C03662=1154.283,339.501,-77.807,-176.527,8.860,148.763
C03663=1154.278,339.780,-77.845,-176.524,8.864,148.763
C03664=1154.274,340.061,-77.883,-176.521,8.869,148.763
C03665=1154.269,340.309,-77.916,-176.518,8.873,148.764
C03666=1154.266,340.556,-77.950,-176.516,8.876,148.764
C03667=1154.261,340.804,-77.983,-176.513,8.880,148.764
C03668=1154.257,341.051,-78.016,-176.510,8.883,148.764
C03669=1154.254,341.299,-78.051,-176.508,8.887,148.764
C03670=1154.249,341.547,-78.084,-176.505,8.891,148.765
C03671=1154.245,341.795,-78.118,-176.503,8.894,148.765
C03672=1154.241,342.042,-78.151,-176.500,8.898,148.765
C03673=1154.237,342.290,-78.185,-176.498,8.902,148.766
C03674=1154.234,342.537,-78.219,-176.495,8.906,148.766
C03675=1154.229,342.786,-78.253,-176.493,8.909,148.766
C03676=1154.225,343.033,-78.286,-176.491,8.912,148.766
C03677=1154.221,343.280,-78.320,-176.488,8.916,148.767
C03678=1154.217,343.528,-78.353,-176.485,8.920,148.767
C03679=1154.213,343.776,-78.388,-176.483,8.924,148.767
C03680=1154.209,344.024,-78.421,-176.481,8.927,148.767
C03681=1154.205,344.271,-78.455,-176.478,8.931,148.768
C03682=1154.200,344.519,-78.488,-176.475,8.935,148.768
C03683=1154.197,344.767,-78.523,-176.473,8.939,148.768
C03684=1154.193,345.014,-78.557,-176.470,8.942,148.768
C03685=1154.188,345.262,-78.590,-176.468,8.945,148.769
C03686=1154.185,345.510,-78.624,-176.465,8.950,148.769
C03687=1154.181,345.758,-78.658,-176.463,8.953,148.769
C03688=1154.176,346.005,-78.692,-176.460,8.957,148.769
C03689=1154.172,346.252,-78.726,-176.458,8.960,148.770
C03690=1154.169,346.501,-78.760,-176.455,8.965,148.770
C03691=1154.164,346.748,-78.794,-176.453,8.968,148.770
C03692=1154.160,346.996,-78.827,-176.450,8.972,148.771
C03693=1154.157,347.243,-78.861,-176.448,8.975,148.771
C03694=1154.152,347.491,-78.896,-176.445,8.980,148.771
C03695=1154.148,347.738,-78.930,-176.443,8.983,148.771
C03696=1154.144,347.987,-78.964,-176.440,8.987,148.771
C03697=1154.140,348.234,-78.998,-176.438,8.991,148.772
C03698=1154.137,348.481,-79.032,-176.435,8.995,148.772
C03699=1154.133,348.729,-79.066,-176.433,8.998,148.772
C03700=1154.128,348.977,-79.100,-176.430,9.001,148.773
C03701=1154.124,349.224,-79.134,-176.428,9.006,148.773
C03702=1154.121,349.472,-79.168,-176.426,9.009,148.773
C03703=1154.116,349.719,-79.203,-176.423,9.013,148.773
C03704=1154.113,349.967,-79.237,-176.420,9.016,148.774
C03705=1154.108,350.215,-79.271,-176.417,9.020,148.774
C03706=1154.104,350.462,-79.305,-176.416,9.024,148.774
C03707=1154.100,350.711,-79.339,-176.413,9.028,148.775
C03708=1154.096,350.958,-79.373,-176.410,9.031,148.775
C03709=1154.092,351.205,-79.408,-176.407,9.035,148.775
C03710=1154.089,351.453,-79.442,-176.406,9.039,148.775
C03711=1154.084,351.700,-79.476,-176.403,9.043,148.776
C03712=1154.081,351.948,-79.511,-176.400,9.046,148.776
C03713=1154.076,352.196,-79.545,-176.398,9.050,148.776
C03714=1154.073,352.443,-79.579,-176.396,9.054,148.777
C03715=1154.068,352.691,-79.614,-176.393,9.058,148.777
C03716=1154.064,352.939,-79.649,-176.390,9.061,148.777
C03717=1154.061,353.186,-79.683,-176.388,9.066,148.778
C03718=1154.056,353.433,-79.717,-176.386,9.069,148.778
C03719=1154.053,353.681,-79.751,-176.383,9.073,148.778
C03720=1154.048,353.929,-79.786,-176.380,9.077,148.778
C03721=1154.044,354.177,-79.821,-176.378,9.081,148.779
C03722=1154.040,354.424,-79.854,-176.375,9.085,148.779
C03723=1154.036,354.672,-79.889,-176.373,9.088,148.779
C03724=1154.032,354.919,-79.924,-176.370,9.093,148.780
C03725=1154.029,355.167,-79.959,-176.368,9.096,148.780
C03726=1154.024,355.414,-79.993,-176.365,9.100,148.780
C03727=1154.020,355.662,-80.028,-176.363,9.104,148.781
C03728=1154.017,355.909,-80.062,-176.360,9.108,148.781
C03729=1154.013,356.157,-80.097,-176.358,9.111,148.781
C03730=1154.008,356.404,-80.132,-176.355,9.115,148.781
C03731=1154.005,356.652,-80.166,-176.353,9.119,148.782
C03732=1154.001,356.900,-80.201,-176.350,9.123,148.782
C03733=1153.997,357.147,-80.236,-176.348,9.126,148.782
C03734=1153.993,357.395,-80.271,-176.345,9.130,148.783
C03735=1153.989,357.642,-80.305,-176.343,9.135,148.783
C03736=1153.985,357.890,-80.340,-176.341,9.138,148.783
C03737=1153.981,358.137,-80.375,-176.338,9.142,148.784
C03738=1153.977,358.385,-80.410,-176.335,9.146,148.784
C03739=1153.973,358.632,-80.444,-176.333,9.150,148.784
C03740=1153.969,358.880,-80.479,-176.331,9.153,148.784
C03741=1153.965,359.128,-80.514,-176.328,9.157,148.785
C03742=1153.961,359.375,-80.549,-176.325,9.162,148.785
C03743=1153.957,359.623,-80.584,-176.323,9.165,148.785
C03744=1153.954,359.869,-80.619,-176.320,9.169,148.786
C03745=1153.950,360.117,-80.653,-176.318,9.173,148.786
C03746=1153.946,360.366,-80.688,-176.315,9.177,148.786
C03747=1153.941,360.612,-80.723,-176.312,9.181,148.787
C03748=1153.937,360.860,-80.758,-176.311,9.184,148.787
C03749=1153.934,361.108,-80.794,-176.308,9.189,148.787
C03750=1153.929,361.355,-80.828,-176.305,9.193,148.788
C03751=1153.926,361.603,-80.863,-176.303,9.196,148.788
C03752=1153.923,361.850,-80.899,-176.300,9.200,148.788
C03753=1153.918,362.098,-80.933,-176.297,9.205,148.789
C03754=1153.914,362.345,-80.969,-176.295,9.208,148.789
C03755=1153.910,362.593,-81.004,-176.292,9.212,148.789
C03756=1153.906,362.840,-81.039,-176.290,9.217,148.790
C03757=1153.902,363.087,-81.074,-176.287,9.220,148.790
C03758=1153.899,363.336,-81.109,-176.285,9.224,148.790
C03759=1153.894,363.582,-81.144,-176.282,9.228,148.791
C03760=1153.891,363.830,-81.180,-176.280,9.232,148.791
C03761=1153.887,364.078,-81.215,-176.277,9.236,148.791
C03762=1153.882,364.325,-81.250,-176.274,9.240,148.792
C03763=1153.879,364.572,-81.285,-176.273,9.244,148.792
C03764=1153.875,364.820,-81.320,-176.270,9.248,148.792
C03765=1153.870,365.103,-81.360,-176.267,9.252,148.793
C03766=1153.866,365.386,-81.401,-176.264,9.257,148.793
C03767=1153.862,365.669,-81.442,-176.261,9.261,148.794
C03768=1153.857,365.952,-81.481,-176.258,9.266,148.794
C03769=1153.853,366.200,-81.518,-176.256,9.270,148.794
C03770=1153.849,366.447,-81.553,-176.253,9.274,148.795
C03771=1153.845,366.694,-81.588,-176.251,9.278,148.795
C03772=1153.841,366.942,-81.623,-176.249,9.282,148.795
C03773=1153.837,367.190,-81.659,-176.246,9.286,148.796
C03774=1153.834,367.437,-81.694,-176.244,9.290,148.796
C03775=1153.829,367.684,-81.729,-176.241,9.294,148.796
C03776=1153.826,367.931,-81.765,-176.238,9.298,148.797
C03777=1153.822,368.179,-81.801,-176.237,9.302,148.797
C03778=1153.818,368.427,-81.837,-176.234,9.306,148.798
C03779=1153.814,368.674,-81.872,-176.231,9.310,148.798
C03780=1153.810,368.921,-81.907,-176.229,9.314,148.798
C03781=1153.806,369.168,-81.943,-176.227,9.318,148.799
C03782=1153.802,369.416,-81.979,-176.224,9.322,148.799
C03783=1153.799,369.663,-82.014,-176.222,9.326,148.800
C03784=1153.794,369.911,-82.050,-176.220,9.330,148.800
C03785=1153.791,370.159,-82.086,-176.218,9.334,148.801
C03786=1153.786,370.406,-82.121,-176.215,9.338,148.801
C03787=1153.783,370.653,-82.156,-176.213,9.343,148.801
C03788=1153.778,370.901,-82.193,-176.211,9.346,148.802
C03789=1153.775,371.148,-82.228,-176.208,9.350,148.802
C03790=1153.771,371.395,-82.264,-176.206,9.354,148.803
C03791=1153.768,371.643,-82.300,-176.204,9.358,148.803
C03792=1153.763,371.891,-82.336,-176.201,9.363,148.804
C03793=1153.759,372.137,-82.371,-176.200,9.367,148.804
C03794=1153.755,372.385,-82.407,-176.197,9.371,148.805
C03795=1153.752,372.632,-82.442,-176.195,9.375,148.805
C03796=1153.748,372.880,-82.479,-176.193,9.379,148.806
C03797=1153.744,373.127,-82.515,-176.191,9.383,148.806
C03798=1153.740,373.375,-82.550,-176.188,9.387,148.806
C03799=1153.736,373.622,-82.586,-176.187,9.391,148.807
C03800=1153.733,373.869,-82.623,-176.184,9.395,148.808
C03801=1153.729,374.117,-82.658,-176.183,9.399,148.808
C03802=1153.725,374.365,-82.694,-176.180,9.403,148.808
C03803=1153.720,374.611,-82.730,-176.179,9.407,148.809
C03804=1153.717,374.858,-82.766,-176.177,9.411,148.809
C03805=1153.712,375.106,-82.802,-176.175,9.416,148.810
C03806=1153.709,375.354,-82.838,-176.173,9.419,148.811
C03807=1153.705,375.601,-82.874,-176.171,9.423,148.811
C03808=1153.701,375.848,-82.910,-176.169,9.427,148.812
C03809=1153.698,376.095,-82.946,-176.167,9.431,148.812
C03810=1153.693,376.343,-82.982,-176.165,9.435,148.813
C03811=1153.690,376.590,-83.018,-176.163,9.440,148.813
C03812=1153.686,376.838,-83.055,-176.162,9.444,148.814
C03813=1153.682,377.085,-83.090,-176.161,9.447,148.815
C03814=1153.678,377.332,-83.127,-176.159,9.451,148.815
C03815=1153.674,377.580,-83.163,-176.157,9.456,148.816
C03816=1153.670,377.827,-83.200,-176.155,9.460,148.816
C03817=1153.666,378.075,-83.235,-176.154,9.464,148.817
C03818=1153.662,378.322,-83.272,-176.152,9.467,148.818
C03819=1153.659,378.569,-83.308,-176.151,9.471,148.818
C03820=1153.655,378.816,-83.344,-176.149,9.475,148.819
C03821=1153.651,379.064,-83.380,-176.148,9.479,148.819
C03822=1153.647,379.311,-83.417,-176.146,9.483,148.820
C03823=1153.643,379.559,-83.452,-176.145,9.487,148.821
C03824=1153.639,379.806,-83.489,-176.144,9.491,148.821
C03825=1153.635,380.053,-83.525,-176.142,9.495,148.822
C03826=1153.631,380.300,-83.562,-176.141,9.499,148.823
C03827=1153.628,380.547,-83.598,-176.139,9.503,148.823
C03828=1153.623,380.795,-83.634,-176.139,9.506,148.824
C03829=1153.620,381.042,-83.670,-176.137,9.510,148.825
C03830=1153.616,381.290,-83.706,-176.136,9.514,148.826
C03831=1153.612,381.537,-83.743,-176.136,9.517,148.826
C03832=1153.608,381.784,-83.780,-176.134,9.522,148.827
C03833=1153.604,382.032,-83.816,-176.133,9.525,148.828
C03834=1153.601,382.279,-83.852,-176.133,9.529,148.828
C03835=1153.597,382.527,-83.889,-176.132,9.533,148.829
C03836=1153.594,382.773,-83.925,-176.131,9.536,148.830
C03837=1153.589,383.021,-83.962,-176.130,9.540,148.830
C03838=1153.585,383.268,-83.998,-176.129,9.544,148.831
C03839=1153.582,383.515,-84.035,-176.129,9.547,148.832
C03840=1153.577,383.763,-84.071,-176.128,9.551,148.833
C03841=1153.573,384.010,-84.108,-176.127,9.555,148.834
C03842=1153.570,384.257,-84.144,-176.127,9.558,148.834
C03843=1153.566,384.504,-84.181,-176.126,9.561,148.835
C03844=1153.562,384.752,-84.216,-176.126,9.565,148.836
C03845=1153.558,384.999,-84.253,-176.125,9.568,148.837
C03846=1153.554,385.246,-84.290,-176.125,9.572,148.837
C03847=1153.551,385.494,-84.327,-176.124,9.575,148.838
C03848=1153.547,385.741,-84.364,-176.124,9.579,148.839
C03849=1153.543,385.989,-84.400,-176.124,9.582,148.840
C03850=1153.539,386.236,-84.436,-176.123,9.585,148.841
C03851=1153.535,386.483,-84.473,-176.124,9.588,148.842
C03852=1153.531,386.730,-84.510,-176.123,9.592,148.842
C03853=1153.528,386.977,-84.546,-176.123,9.595,148.843
C03854=1153.523,387.225,-84.582,-176.124,9.598,148.844
C03855=1153.519,387.472,-84.619,-176.123,9.601,148.845
C03856=1153.517,387.720,-84.656,-176.124,9.604,148.846
C03857=1153.513,387.967,-84.692,-176.123,9.608,148.846
C03858=1153.508,388.214,-84.729,-176.124,9.610,148.847
C03859=1153.504,388.461,-84.766,-176.124,9.613,148.848
C03860=1153.501,388.708,-84.802,-176.124,9.617,148.849
C03861=1153.497,388.956,-84.839,-176.124,9.620,148.850
C03862=1153.492,389.203,-84.875,-176.124,9.622,148.851
C03863=1153.490,389.451,-84.912,-176.125,9.625,148.851
C03864=1153.486,389.698,-84.949,-176.125,9.628,148.852
C03865=1153.482,389.945,-84.986,-176.126,9.630,148.853
C03866=1153.478,390.192,-85.022,-176.126,9.633,148.854
C03867=1153.474,390.439,-85.059,-176.127,9.636,148.855
C03868=1153.470,390.686,-85.096,-176.127,9.639,148.856
C03869=1153.466,390.973,-85.138,-176.127,9.643,148.857
C03870=1153.461,391.260,-85.181,-176.128,9.646,148.858
C03871=1153.456,391.545,-85.223,-176.128,9.648,148.858
C03872=1153.453,391.832,-85.265,-176.129,9.652,148.860
C03873=1153.449,392.079,-85.302,-176.129,9.654,148.860
C03874=1153.445,392.326,-85.339,-176.130,9.657,148.861
C03875=1153.441,392.573,-85.376,-176.131,9.659,148.862
C03876=1153.437,392.820,-85.412,-176.132,9.662,148.863
C03877=1153.434,393.068,-85.449,-176.132,9.665,148.864
C03878=1153.430,393.315,-85.486,-176.133,9.667,148.864
C03879=1153.426,393.562,-85.523,-176.133,9.670,148.865
C03880=1153.422,393.809,-85.559,-176.134,9.672,148.866
C03881=1153.418,394.056,-85.596,-176.135,9.674,148.867
C03882=1153.414,394.304,-85.633,-176.136,9.676,148.868
C03883=1153.410,394.552,-85.670,-176.136,9.679,148.869
C03884=1153.407,394.799,-85.706,-176.137,9.681,148.869
C03885=1153.403,395.046,-85.742,-176.138,9.684,148.870
C03886=1153.399,395.293,-85.779,-176.139,9.686,148.871
C03887=1153.395,395.541,-85.816,-176.139,9.689,148.872
C03888=1153.391,395.787,-85.852,-176.140,9.691,148.873
C03889=1153.387,396.035,-85.889,-176.141,9.693,148.874
C03890=1153.384,396.283,-85.926,-176.142,9.696,148.875
C03891=1153.379,396.530,-85.963,-176.143,9.698,148.875
C03892=1153.376,396.777,-86.000,-176.144,9.699,148.876
C03893=1153.372,397.024,-86.036,-176.144,9.702,148.877
C03894=1153.368,397.271,-86.073,-176.145,9.704,148.878
C03895=1153.364,397.518,-86.110,-176.146,9.706,148.879
C03896=1153.360,397.766,-86.147,-176.147,9.708,148.879
C03897=1153.357,398.013,-86.184,-176.148,9.711,148.880
C03898=1153.353,398.260,-86.220,-176.149,9.713,148.881
C03899=1153.349,398.507,-86.257,-176.150,9.715,148.882
C03900=1153.345,398.755,-86.294,-176.151,9.717,148.882
C03901=1153.341,399.001,-86.330,-176.152,9.719,148.883
C03902=1153.338,399.249,-86.368,-176.153,9.721,148.884
C03903=1153.334,399.497,-86.405,-176.153,9.723,148.885
C03904=1153.330,399.744,-86.441,-176.154,9.726,148.886
C03905=1153.326,399.991,-86.478,-176.155,9.728,148.887
C03906=1153.322,400.238,-86.515,-176.156,9.730,148.887
C03907=1153.318,400.485,-86.551,-176.157,9.732,148.888
C03908=1153.315,400.733,-86.589,-176.158,9.734,148.889
C03909=1153.311,400.980,-86.625,-176.159,9.735,148.889
C03910=1153.307,401.227,-86.662,-176.160,9.737,148.890
C03911=1153.303,401.475,-86.698,-176.161,9.739,148.891
C03912=1153.299,401.722,-86.735,-176.162,9.741,148.892
C03913=1153.295,401.969,-86.772,-176.163,9.743,148.893
C03914=1153.292,402.217,-86.808,-176.163,9.745,148.893
C03915=1153.288,402.464,-86.845,-176.165,9.747,148.894
C03916=1153.284,402.711,-86.882,-176.166,9.749,148.895
C03917=1153.280,402.958,-86.919,-176.166,9.751,148.896
C03918=1153.275,403.205,-86.956,-176.167,9.753,148.896
C03919=1153.272,403.452,-86.992,-176.168,9.755,148.897
C03920=1153.269,403.700,-87.029,-176.169,9.757,148.898
C03921=1153.265,403.947,-87.066,-176.170,9.759,148.899
C03922=1153.260,404.195,-87.103,-176.171,9.761,148.899
C03923=1153.257,404.441,-87.139,-176.172,9.762,148.900
C03924=1153.253,404.689,-87.176,-176.172,9.764,148.901
C03925=1153.249,404.936,-87.213,-176.174,9.766,148.902
C03926=1153.245,405.184,-87.250,-176.174,9.768,148.902
C03927=1153.241,405.431,-87.287,-176.175,9.770,148.903
C03928=1153.238,405.678,-87.323,-176.176,9.772,148.904
C03929=1153.234,405.925,-87.360,-176.177,9.773,148.904
C03930=1153.230,406.172,-87.397,-176.178,9.776,148.905
C03931=1153.226,406.419,-87.434,-176.179,9.777,148.906
C03932=1153.222,406.667,-87.471,-176.180,9.779,148.907
C03933=1153.219,406.914,-87.507,-176.180,9.781,148.907
C03934=1153.215,407.161,-87.544,-176.181,9.783,148.908
C03935=1153.211,407.409,-87.581,-176.182,9.785,148.909
C03936=1153.207,407.656,-87.618,-176.183,9.787,148.909
C03937=1153.203,407.903,-87.654,-176.183,9.788,148.910
C03938=1153.200,408.151,-87.691,-176.184,9.790,148.911
C03939=1153.196,408.398,-87.728,-176.185,9.792,148.912
C03940=1153.191,408.645,-87.765,-176.186,9.794,148.912
C03941=1153.187,408.892,-87.802,-176.187,9.796,148.913
C03942=1153.184,409.139,-87.838,-176.187,9.797,148.913
C03943=1153.180,409.386,-87.875,-176.188,9.800,148.914
C03944=1153.176,409.634,-87.912,-176.189,9.801,148.915
C03945=1153.172,409.881,-87.949,-176.190,9.803,148.916
C03946=1153.168,410.128,-87.986,-176.190,9.805,148.916
C03947=1153.165,410.375,-88.022,-176.191,9.807,148.917
C03948=1153.161,410.622,-88.059,-176.192,9.808,148.918
C03949=1153.157,410.870,-88.096,-176.193,9.810,148.918
C03950=1153.153,411.118,-88.133,-176.194,9.812,148.919
C03951=1153.149,411.365,-88.170,-176.194,9.814,148.920
C03952=1153.146,411.612,-88.206,-176.195,9.816,148.920
C03953=1153.142,411.859,-88.243,-176.196,9.817,148.921
C03954=1153.138,412.106,-88.280,-176.196,9.819,148.922
C03955=1153.134,412.354,-88.317,-176.196,9.822,148.922
C03956=1153.130,412.601,-88.354,-176.197,9.823,148.923
C03957=1153.127,412.848,-88.390,-176.198,9.825,148.924
C03958=1153.123,413.095,-88.427,-176.199,9.827,148.924
C03959=1153.118,413.342,-88.464,-176.199,9.829,148.925
C03960=1153.114,413.590,-88.501,-176.200,9.830,148.925
C03961=1153.111,413.837,-88.538,-176.201,9.832,148.926
C03962=1153.107,414.084,-88.574,-176.202,9.834,148.927
C03963=1153.103,414.332,-88.611,-176.202,9.836,148.928
C03964=1153.099,414.579,-88.648,-176.203,9.838,148.928
C03965=1153.095,414.826,-88.685,-176.203,9.840,148.929
C03966=1153.093,415.073,-88.722,-176.203,9.842,148.929
C03967=1153.090,415.320,-88.759,-176.204,9.843,148.930
C03968=1153.088,415.568,-88.795,-176.205,9.845,148.931
C03969=1153.087,415.777,-88.826,-176.205,9.847,148.931
C03970=1153.087,415.987,-88.857,-176.206,9.848,148.932
C03971=1153.087,416.196,-88.888,-176.206,9.850,148.932
C03972=1153.087,416.407,-88.919,-176.207,9.852,148.933
C03973=1153.091,416.825,-88.981,-176.207,9.854,148.934
C03974=1153.097,417.243,-89.041,-176.209,9.857,148.935
C03975=1152.676,417.245,-89.089,-176.211,9.868,148.938
C03976=1152.673,417.034,-89.059,-176.210,9.867,148.938
C03977=1152.670,416.824,-89.028,-176.210,9.865,148.937
C03978=1152.669,416.613,-88.997,-176.209,9.864,148.937
C03979=1152.667,416.401,-88.966,-176.209,9.862,148.936
C03980=1152.666,416.190,-88.935,-176.209,9.861,148.936
C03981=1152.666,415.979,-88.904,-176.208,9.859,148.935
C03982=1152.666,415.767,-88.873,-176.208,9.858,148.935
C03983=1152.667,415.556,-88.841,-176.207,9.856,148.934
C03984=1152.669,415.309,-88.805,-176.207,9.854,148.934
C03985=1152.672,415.062,-88.768,-176.206,9.853,148.933
C03986=1152.675,414.815,-88.731,-176.206,9.851,148.932
C03987=1152.679,414.567,-88.695,-176.205,9.849,148.932
C03988=1152.683,414.320,-88.658,-176.204,9.847,148.931
C03989=1152.687,414.073,-88.621,-176.204,9.845,148.930
C03990=1152.690,413.825,-88.584,-176.203,9.843,148.930
C03991=1152.694,413.578,-88.547,-176.203,9.841,148.929
C03992=1152.698,413.331,-88.511,-176.202,9.839,148.928
C03993=1152.702,413.084,-88.474,-176.201,9.838,148.928
C03994=1152.706,412.837,-88.437,-176.200,9.836,148.927
C03995=1152.710,412.589,-88.400,-176.200,9.834,148.926
C03996=1152.713,412.342,-88.363,-176.199,9.832,148.926
C03997=1152.717,412.095,-88.326,-176.198,9.831,148.925
C03998=1152.721,411.847,-88.290,-176.198,9.829,148.924
C03999=1152.725,411.600,-88.253,-176.197,9.827,148.924
C04000=1152.729,411.353,-88.216,-176.197,9.825,148.923
C04001=1152.733,411.105,-88.179,-176.196,9.822,148.922
C04002=1152.736,410.858,-88.142,-176.195,9.821,148.922
C04003=1152.740,410.611,-88.106,-176.195,9.819,148.921
C04004=1152.744,410.364,-88.069,-176.194,9.817,148.920
C04005=1152.748,410.117,-88.032,-176.193,9.815,148.920
C04006=1152.752,409.869,-87.995,-176.192,9.814,148.919
C04007=1152.755,409.622,-87.958,-176.191,9.812,148.918
C04008=1152.759,409.375,-87.922,-176.191,9.810,148.918
C04009=1152.763,409.128,-87.885,-176.190,9.808,148.917
C04010=1152.768,408.880,-87.848,-176.189,9.806,148.916
C04011=1152.772,408.633,-87.811,-176.188,9.804,148.915
C04012=1152.774,408.386,-87.774,-176.188,9.803,148.915
C04013=1152.778,408.138,-87.737,-176.187,9.801,148.914
C04014=1152.783,407.891,-87.701,-176.186,9.799,148.914
C04015=1152.787,407.644,-87.664,-176.185,9.797,148.913
C04016=1152.790,407.397,-87.627,-176.184,9.795,148.912
C04017=1152.794,407.149,-87.590,-176.184,9.794,148.911
C04018=1152.798,406.902,-87.553,-176.183,9.791,148.911
C04019=1152.802,406.655,-87.517,-176.182,9.790,148.910
C04020=1152.806,406.408,-87.480,-176.181,9.788,148.909
C04021=1152.809,406.161,-87.443,-176.180,9.786,148.908
C04022=1152.813,405.914,-87.407,-176.179,9.784,148.908
C04023=1152.817,405.666,-87.369,-176.178,9.782,148.907
C04024=1152.821,405.419,-87.332,-176.177,9.781,148.906
C04025=1152.825,405.171,-87.296,-176.176,9.779,148.906
C04026=1152.828,404.925,-87.259,-176.175,9.777,148.905
C04027=1152.832,404.677,-87.222,-176.175,9.776,148.904
C04028=1152.836,404.430,-87.186,-176.173,9.774,148.903
C04029=1152.840,404.182,-87.148,-176.173,9.772,148.903
C04030=1152.844,403.935,-87.112,-176.172,9.770,148.902
C04031=1152.847,403.688,-87.075,-176.171,9.768,148.901
C04032=1152.852,403.441,-87.038,-176.170,9.766,148.900
C04033=1152.856,403.194,-87.002,-176.169,9.764,148.900
C04034=1152.859,402.946,-86.964,-176.168,9.762,148.899
C04035=1152.862,402.699,-86.928,-176.167,9.760,148.898
C04036=1152.867,402.452,-86.891,-176.166,9.758,148.898
C04037=1152.871,402.205,-86.854,-176.165,9.756,148.897
C04038=1152.875,401.957,-86.817,-176.164,9.754,148.896
C04039=1152.879,401.710,-86.781,-176.163,9.752,148.895
C04040=1152.882,401.463,-86.744,-176.163,9.751,148.895
C04041=1152.886,401.215,-86.707,-176.162,9.749,148.894
C04042=1152.890,400.968,-86.670,-176.160,9.747,148.893
C04043=1152.894,400.721,-86.633,-176.160,9.745,148.892
C04044=1152.898,400.474,-86.597,-176.159,9.742,148.891
C04045=1152.901,400.227,-86.560,-176.158,9.740,148.890
C04046=1152.905,399.979,-86.523,-176.157,9.738,148.890
C04047=1152.909,399.732,-86.486,-176.156,9.736,148.889
C04048=1152.913,399.485,-86.449,-176.155,9.734,148.888
C04049=1152.916,399.238,-86.413,-176.154,9.732,148.888
C04050=1152.920,398.991,-86.376,-176.153,9.730,148.887
C04051=1152.925,398.744,-86.339,-176.152,9.728,148.886
C04052=1152.928,398.496,-86.302,-176.151,9.726,148.885
C04053=1152.932,398.248,-86.265,-176.151,9.724,148.884
C04054=1152.935,398.002,-86.229,-176.150,9.721,148.883
C04055=1152.940,397.754,-86.192,-176.149,9.719,148.883
C04056=1152.944,397.507,-86.155,-176.148,9.717,148.882
C04057=1152.948,397.260,-86.118,-176.147,9.716,148.881
C04058=1152.951,397.012,-86.082,-176.146,9.713,148.880
C04059=1152.955,396.765,-86.045,-176.145,9.711,148.879
C04060=1152.959,396.518,-86.008,-176.144,9.709,148.879
C04061=1152.963,396.271,-85.971,-176.143,9.707,148.878
C04062=1152.967,396.024,-85.934,-176.143,9.704,148.877
C04063=1152.970,395.777,-85.898,-176.142,9.702,148.876
C04064=1152.974,395.529,-85.861,-176.141,9.700,148.875
C04065=1152.978,395.282,-85.824,-176.140,9.697,148.874
C04066=1152.982,395.034,-85.787,-176.139,9.695,148.874
C04067=1152.985,394.788,-85.751,-176.139,9.692,148.873
C04068=1152.989,394.540,-85.714,-176.138,9.690,148.872
C04069=1152.993,394.293,-85.677,-176.137,9.687,148.871
C04070=1152.998,394.046,-85.640,-176.136,9.685,148.870
C04071=1153.000,393.798,-85.604,-176.136,9.682,148.869
C04072=1153.004,393.551,-85.567,-176.135,9.681,148.869
C04073=1153.009,393.303,-85.531,-176.134,9.678,148.868
C04074=1153.013,393.056,-85.494,-176.133,9.676,148.867
C04075=1153.016,392.809,-85.458,-176.133,9.673,148.866
C04076=1153.020,392.562,-85.421,-176.132,9.670,148.865
C04077=1153.024,392.314,-85.384,-176.132,9.668,148.865
C04078=1153.028,392.067,-85.347,-176.131,9.665,148.864
C04079=1153.031,391.820,-85.310,-176.131,9.663,148.863
C04080=1153.035,391.534,-85.267,-176.130,9.660,148.862
C04081=1153.040,391.248,-85.225,-176.129,9.656,148.861
C04082=1153.045,390.961,-85.183,-176.129,9.654,148.860
C04083=1153.049,390.675,-85.140,-176.128,9.651,148.859
C04084=1153.053,390.428,-85.103,-176.127,9.648,148.858
C04085=1153.057,390.181,-85.066,-176.127,9.645,148.857
C04086=1153.060,389.934,-85.030,-176.126,9.642,148.856
C04087=1153.065,389.686,-84.994,-176.127,9.639,148.856
C04088=1153.069,389.439,-84.957,-176.126,9.636,148.855
C04089=1153.072,389.191,-84.920,-176.126,9.633,148.854
C04090=1153.076,388.944,-84.883,-176.126,9.630,148.853
C04091=1153.080,388.697,-84.847,-176.125,9.628,148.852
C04092=1153.084,388.450,-84.810,-176.125,9.625,148.851
C04093=1153.087,388.203,-84.773,-176.125,9.621,148.850
C04094=1153.091,387.956,-84.737,-176.124,9.618,148.850
C04095=1153.096,387.708,-84.700,-176.125,9.615,148.849
C04096=1153.099,387.460,-84.664,-176.124,9.612,148.848
C04097=1153.103,387.213,-84.627,-176.125,9.609,148.847
C04098=1153.107,386.966,-84.590,-176.125,9.606,148.846
C04099=1153.110,386.719,-84.554,-176.125,9.603,148.845
C04100=1153.114,386.472,-84.517,-176.125,9.600,148.845
C04101=1153.118,386.225,-84.480,-176.125,9.596,148.844
C04102=1153.122,385.977,-84.445,-176.125,9.593,148.843
C04103=1153.126,385.730,-84.408,-176.126,9.590,148.842
C04104=1153.130,385.483,-84.371,-176.126,9.587,148.842
C04105=1153.133,385.235,-84.334,-176.126,9.583,148.841
C04106=1153.137,384.988,-84.297,-176.126,9.580,148.840
C04107=1153.141,384.740,-84.261,-176.127,9.576,148.839
C04108=1153.145,384.493,-84.225,-176.127,9.573,148.838
C04109=1153.149,384.246,-84.188,-176.128,9.569,148.838
C04110=1153.153,383.999,-84.151,-176.128,9.566,148.837
C04111=1153.157,383.751,-84.116,-176.129,9.562,148.836
C04112=1153.161,383.504,-84.079,-176.129,9.559,148.835
C04113=1153.165,383.257,-84.042,-176.130,9.555,148.834
C04114=1153.168,383.010,-84.006,-176.131,9.551,148.834
C04115=1153.172,382.762,-83.969,-176.132,9.548,148.833
C04116=1153.175,382.515,-83.933,-176.133,9.544,148.832
C04117=1153.179,382.268,-83.896,-176.133,9.541,148.832
C04118=1153.184,382.020,-83.859,-176.135,9.537,148.831
C04119=1153.187,381.773,-83.824,-176.136,9.532,148.830
C04120=1153.191,381.526,-83.787,-176.137,9.529,148.830
C04121=1153.195,381.279,-83.751,-176.138,9.525,148.829
C04122=1153.199,381.031,-83.714,-176.139,9.521,148.828
C04123=1153.203,380.784,-83.678,-176.140,9.518,148.827
C04124=1153.207,380.536,-83.642,-176.141,9.514,148.827
C04125=1153.211,380.289,-83.605,-176.143,9.510,148.826
C04126=1153.214,380.042,-83.569,-176.144,9.506,148.825
C04127=1153.219,379.794,-83.533,-176.145,9.502,148.825
C04128=1153.222,379.548,-83.497,-176.147,9.498,148.824
C04129=1153.226,379.300,-83.460,-176.148,9.494,148.823
C04130=1153.230,379.053,-83.424,-176.150,9.490,148.823
C04131=1153.234,378.806,-83.387,-176.151,9.486,148.822
C04132=1153.238,378.558,-83.352,-176.152,9.482,148.821
C04133=1153.242,378.311,-83.315,-176.154,9.478,148.821
C04134=1153.245,378.063,-83.279,-176.155,9.474,148.820
C04135=1153.249,377.816,-83.242,-176.157,9.471,148.820
C04136=1153.253,377.569,-83.207,-176.158,9.467,148.819
C04137=1153.257,377.322,-83.170,-176.160,9.462,148.818
C04138=1153.261,377.074,-83.134,-176.162,9.458,148.818
C04139=1153.265,376.827,-83.098,-176.163,9.454,148.817
C04140=1153.269,376.579,-83.062,-176.165,9.451,148.817
C04141=1153.273,376.332,-83.026,-176.167,9.446,148.816
C04142=1153.276,376.085,-82.990,-176.169,9.442,148.815
C04143=1153.280,375.837,-82.954,-176.171,9.439,148.815
C04144=1153.284,375.590,-82.917,-176.173,9.434,148.814
C04145=1153.288,375.342,-82.882,-176.175,9.430,148.814
C04146=1153.292,375.095,-82.846,-176.176,9.427,148.813
C04147=1153.296,374.848,-82.809,-176.179,9.422,148.813
C04148=1153.299,374.600,-82.774,-176.180,9.419,148.812
C04149=1153.304,374.352,-82.738,-176.182,9.414,148.812
C04150=1153.307,374.106,-82.701,-176.184,9.410,148.811
C04151=1153.311,373.858,-82.665,-176.187,9.406,148.811
C04152=1153.315,373.610,-82.630,-176.188,9.402,148.810
C04153=1153.319,373.364,-82.594,-176.191,9.398,148.810
C04154=1153.323,373.116,-82.558,-176.193,9.394,148.809
C04155=1153.327,372.869,-82.522,-176.195,9.390,148.809
C04156=1153.331,372.621,-82.487,-176.197,9.386,148.808
C04157=1153.334,372.374,-82.451,-176.199,9.381,148.808
C04158=1153.338,372.127,-82.414,-176.201,9.378,148.807
C04159=1153.342,371.879,-82.379,-176.203,9.373,148.807
C04160=1153.346,371.632,-82.343,-176.205,9.370,148.806
C04161=1153.350,371.384,-82.307,-176.208,9.365,148.806
C04162=1153.354,371.137,-82.272,-176.210,9.361,148.806
C04163=1153.358,370.889,-82.236,-176.213,9.358,148.805
C04164=1153.361,370.643,-82.200,-176.215,9.353,148.805
C04165=1153.366,370.395,-82.164,-176.217,9.350,148.804
C04166=1153.370,370.147,-82.128,-176.219,9.345,148.804
C04167=1153.373,369.900,-82.093,-176.222,9.341,148.803
C04168=1153.377,369.652,-82.057,-176.224,9.337,148.803
C04169=1153.381,369.406,-82.022,-176.226,9.333,148.803
C04170=1153.385,369.158,-81.986,-176.229,9.329,148.802
C04171=1153.389,368.910,-81.950,-176.231,9.325,148.802
C04172=1153.393,368.663,-81.915,-176.234,9.321,148.801
C04173=1153.396,368.415,-81.879,-176.236,9.317,148.801
C04174=1153.401,368.168,-81.844,-176.238,9.313,148.801
C04175=1153.404,367.921,-81.808,-176.241,9.309,148.800
C04176=1153.409,367.673,-81.772,-176.244,9.305,148.800
C04177=1153.412,367.426,-81.737,-176.246,9.301,148.800
C04178=1153.416,367.178,-81.701,-176.248,9.297,148.799
C04179=1153.421,366.931,-81.667,-176.251,9.292,148.799
C04180=1153.424,366.683,-81.631,-176.253,9.289,148.798
C04181=1153.428,366.436,-81.596,-176.256,9.285,148.798
C04182=1153.432,366.188,-81.560,-176.258,9.280,148.798
C04183=1153.436,365.941,-81.525,-176.261,9.277,148.797
C04184=1153.440,365.658,-81.484,-176.264,9.272,148.797
C04185=1153.445,365.375,-81.443,-176.266,9.267,148.796
C04186=1153.449,365.092,-81.403,-176.269,9.263,148.796
C04187=1153.453,364.809,-81.363,-176.272,9.258,148.796
C04188=1153.458,364.561,-81.328,-176.275,9.254,148.795
C04189=1153.462,364.314,-81.293,-176.277,9.250,148.795
C04190=1153.465,364.066,-81.257,-176.280,9.246,148.795
C04191=1153.469,363.818,-81.222,-176.283,9.242,148.794
C04192=1153.474,363.572,-81.187,-176.285,9.239,148.794
C04193=1153.477,363.324,-81.152,-176.287,9.235,148.794
C04194=1153.481,363.076,-81.117,-176.290,9.230,148.793
C04195=1153.486,362.829,-81.082,-176.292,9.227,148.793
C04196=1153.489,362.582,-81.046,-176.295,9.223,148.793
C04197=1153.493,362.333,-81.011,-176.298,9.218,148.792
C04198=1153.497,362.087,-80.976,-176.300,9.215,148.792
C04199=1153.501,361.839,-80.940,-176.302,9.211,148.792
C04200=1153.505,361.591,-80.906,-176.305,9.207,148.791
C04201=1153.509,361.345,-80.871,-176.308,9.203,148.791
C04202=1153.513,361.096,-80.836,-176.310,9.199,148.791
C04203=1153.516,360.849,-80.801,-176.312,9.196,148.790
C04204=1153.521,360.602,-80.766,-176.315,9.192,148.790
C04205=1153.524,360.354,-80.731,-176.318,9.187,148.790
C04206=1153.528,360.106,-80.696,-176.320,9.184,148.790
C04207=1153.533,359.859,-80.661,-176.323,9.180,148.789
C04208=1153.536,359.611,-80.626,-176.325,9.175,148.789
C04209=1153.540,359.365,-80.591,-176.328,9.172,148.789
C04210=1153.544,359.116,-80.556,-176.330,9.168,148.788
C04211=1153.548,358.868,-80.522,-176.333,9.164,148.788
C04212=1153.552,358.621,-80.486,-176.335,9.160,148.788
C04213=1153.556,358.374,-80.452,-176.338,9.156,148.787
C04214=1153.560,358.126,-80.418,-176.340,9.153,148.787
C04215=1153.564,357.879,-80.382,-176.343,9.149,148.787
C04216=1153.568,357.631,-80.347,-176.345,9.145,148.786
C04217=1153.572,357.383,-80.313,-176.348,9.141,148.786
C04218=1153.575,357.136,-80.278,-176.350,9.138,148.786
C04219=1153.580,356.889,-80.243,-176.353,9.133,148.785
C04220=1153.584,356.640,-80.209,-176.356,9.129,148.785
C04221=1153.587,356.394,-80.174,-176.358,9.126,148.785
C04222=1153.591,356.146,-80.139,-176.360,9.121,148.784
C04223=1153.596,355.898,-80.105,-176.363,9.118,148.784
C04224=1153.600,355.650,-80.070,-176.366,9.114,148.784
C04225=1153.604,355.403,-80.036,-176.368,9.110,148.784
C04226=1153.607,355.156,-80.000,-176.370,9.106,148.783
C04227=1153.612,354.908,-79.966,-176.373,9.103,148.783
C04228=1153.615,354.660,-79.932,-176.375,9.099,148.783
C04229=1153.620,354.413,-79.897,-176.378,9.095,148.782
C04230=1153.624,354.165,-79.862,-176.380,9.091,148.782
C04231=1153.628,353.918,-79.829,-176.383,9.088,148.782
C04232=1153.631,353.670,-79.794,-176.385,9.084,148.781
C04233=1153.635,353.423,-79.760,-176.388,9.080,148.781
C04234=1153.639,353.175,-79.724,-176.390,9.076,148.781
C04235=1153.644,352.928,-79.690,-176.393,9.072,148.780
C04236=1153.647,352.680,-79.656,-176.395,9.069,148.780
C04237=1153.651,352.432,-79.621,-176.398,9.065,148.780
C04238=1153.655,352.185,-79.587,-176.400,9.061,148.780
C04239=1153.659,351.937,-79.552,-176.403,9.057,148.779
C04240=1153.662,351.689,-79.518,-176.405,9.054,148.779
C04241=1153.667,351.442,-79.484,-176.408,9.049,148.779
C04242=1153.672,351.194,-79.450,-176.410,9.046,148.778
C04243=1153.675,350.946,-79.416,-176.413,9.042,148.778
C04244=1153.680,350.699,-79.381,-176.415,9.038,148.778
C04245=1153.683,350.451,-79.347,-176.418,9.034,148.778
C04246=1153.687,350.204,-79.313,-176.420,9.031,148.777
C04247=1153.691,349.956,-79.279,-176.423,9.027,148.777
C04248=1153.695,349.708,-79.244,-176.425,9.023,148.777
C04249=1153.699,349.461,-79.210,-176.428,9.019,148.777
C04250=1153.703,349.213,-79.175,-176.430,9.016,148.776
C04251=1153.707,348.965,-79.142,-176.433,9.012,148.776
C04252=1153.711,348.718,-79.108,-176.435,9.008,148.776
C04253=1153.715,348.470,-79.073,-176.438,9.004,148.775
C04254=1153.719,348.223,-79.039,-176.440,9.001,148.775
C04255=1153.724,347.975,-79.006,-176.443,8.997,148.775
C04256=1153.727,347.727,-78.971,-176.445,8.993,148.775
C04257=1153.731,347.480,-78.937,-176.448,8.989,148.774
C04258=1153.735,347.233,-78.903,-176.450,8.986,148.774
C04259=1153.739,346.984,-78.870,-176.453,8.983,148.774
C04260=1153.743,346.737,-78.835,-176.455,8.978,148.773
C04261=1153.747,346.490,-78.801,-176.458,8.975,148.773
C04262=1153.752,346.241,-78.767,-176.460,8.971,148.773
C04263=1153.755,345.994,-78.733,-176.463,8.968,148.773
C04264=1153.759,345.747,-78.699,-176.466,8.964,148.773
C04265=1153.764,345.499,-78.666,-176.468,8.960,148.772
C04266=1153.767,345.251,-78.631,-176.470,8.956,148.772
C04267=1153.771,345.003,-78.598,-176.473,8.953,148.772
C04268=1153.776,344.756,-78.564,-176.476,8.948,148.771
C04269=1153.780,344.507,-78.530,-176.478,8.945,148.771
C04270=1153.783,344.260,-78.496,-176.481,8.941,148.771
C04271=1153.787,344.013,-78.463,-176.483,8.938,148.771
C04272=1153.792,343.765,-78.429,-176.485,8.934,148.770
C04273=1153.795,343.517,-78.395,-176.488,8.930,148.770
C04274=1153.799,343.269,-78.361,-176.490,8.927,148.770
C04275=1153.804,343.021,-78.328,-176.493,8.923,148.770
C04276=1153.808,342.774,-78.294,-176.495,8.919,148.769
C04277=1153.812,342.527,-78.261,-176.498,8.915,148.769
C04278=1153.816,342.279,-78.226,-176.501,8.912,148.769
C04279=1153.820,342.031,-78.193,-176.503,8.908,148.769
C04280=1153.824,341.784,-78.159,-176.505,8.904,148.768
C04281=1153.828,341.536,-78.126,-176.508,8.901,148.768
C04282=1153.832,341.287,-78.092,-176.511,8.897,148.768
C04283=1153.836,341.040,-78.058,-176.513,8.894,148.768
C04284=1153.840,340.793,-78.025,-176.516,8.890,148.767
C04285=1153.845,340.545,-77.991,-176.518,8.886,148.767
C04286=1153.849,340.297,-77.957,-176.521,8.882,148.767
C04287=1153.853,340.050,-77.924,-176.523,8.879,148.767
C04288=1153.857,339.769,-77.886,-176.526,8.875,148.766
C04289=1153.862,339.490,-77.848,-176.529,8.871,148.766
C04290=1153.866,339.209,-77.810,-176.532,8.866,148.766
C04291=1153.871,338.930,-77.773,-176.535,8.862,148.766
C04292=1153.875,338.682,-77.740,-176.537,8.859,148.765
C04293=1153.879,338.434,-77.706,-176.540,8.855,148.765
C04294=1153.882,338.186,-77.673,-176.542,8.852,148.765
C04295=1153.887,337.938,-77.640,-176.545,8.848,148.765
C04296=1153.890,337.691,-77.606,-176.547,8.844,148.764
C04297=1153.895,337.443,-77.572,-176.550,8.841,148.764
C04298=1153.899,337.195,-77.539,-176.552,8.837,148.764
C04299=1153.904,336.947,-77.506,-176.555,8.834,148.764
C04300=1153.908,336.700,-77.473,-176.558,8.830,148.764
C04301=1153.912,336.452,-77.440,-176.560,8.826,148.763
C04302=1153.916,336.204,-77.406,-176.562,8.823,148.763
C04303=1153.920,335.956,-77.373,-176.565,8.819,148.763
C04304=1153.924,335.708,-77.340,-176.567,8.815,148.763
C04305=1153.927,335.461,-77.307,-176.570,8.811,148.762
C04306=1153.931,335.213,-77.274,-176.572,8.808,148.762
C04307=1153.935,334.965,-77.241,-176.575,8.805,148.762
C04308=1153.940,334.717,-77.208,-176.578,8.801,148.762
C04309=1153.944,334.470,-77.175,-176.580,8.797,148.761
C04310=1153.948,334.222,-77.141,-176.583,8.793,148.761
C04311=1153.952,333.974,-77.108,-176.585,8.790,148.761
C04312=1153.956,333.727,-77.075,-176.587,8.787,148.761
C04313=1153.960,333.479,-77.042,-176.590,8.783,148.761
C04314=1153.964,333.231,-77.009,-176.593,8.779,148.760
C04315=1153.968,332.983,-76.976,-176.595,8.776,148.760
C04316=1153.973,332.736,-76.942,-176.598,8.772,148.760
C04317=1153.976,332.488,-76.910,-176.600,8.769,148.760
C04318=1153.980,332.240,-76.877,-176.603,8.765,148.759
C04319=1153.985,331.992,-76.844,-176.605,8.761,148.759
C04320=1153.989,331.744,-76.811,-176.608,8.758,148.759
C04321=1153.993,331.497,-76.778,-176.611,8.754,148.759
C04322=1153.997,331.249,-76.745,-176.613,8.751,148.759
C04323=1154.001,331.001,-76.713,-176.616,8.748,148.759
C04324=1154.005,330.753,-76.680,-176.619,8.744,148.758
C04325=1154.009,330.505,-76.647,-176.621,8.740,148.758
C04326=1154.013,330.258,-76.614,-176.624,8.736,148.758
C04327=1154.018,330.009,-76.581,-176.626,8.733,148.758
C04328=1154.021,329.762,-76.549,-176.628,8.730,148.758
C04329=1154.025,329.514,-76.515,-176.631,8.726,148.757
C04330=1154.030,329.266,-76.483,-176.634,8.722,148.757
C04331=1154.034,329.018,-76.450,-176.636,8.719,148.757
C04332=1154.037,328.771,-76.417,-176.639,8.715,148.757
C04333=1154.042,328.522,-76.385,-176.641,8.712,148.756
C04334=1154.046,328.275,-76.352,-176.643,8.708,148.756
C04335=1154.049,328.027,-76.320,-176.646,8.704,148.756
C04336=1154.054,327.780,-76.287,-176.649,8.701,148.756
C04337=1154.058,327.532,-76.254,-176.651,8.698,148.756
C04338=1154.062,327.284,-76.222,-176.654,8.694,148.755
C04339=1154.066,327.036,-76.189,-176.657,8.691,148.755
C04340=1154.071,326.788,-76.156,-176.659,8.687,148.755
C04341=1154.074,326.540,-76.124,-176.662,8.683,148.755
C04342=1154.078,326.292,-76.091,-176.664,8.680,148.755
C04343=1154.083,326.044,-76.058,-176.666,8.677,148.755
C04344=1154.086,325.796,-76.026,-176.669,8.673,148.754
C04345=1154.091,325.549,-75.994,-176.672,8.669,148.754
C04346=1154.095,325.301,-75.961,-176.674,8.666,148.754
C04347=1154.099,325.053,-75.929,-176.677,8.662,148.754
C04348=1154.103,324.805,-75.896,-176.680,8.659,148.754
C04349=1154.107,324.557,-75.864,-176.682,8.656,148.754
C04350=1154.111,324.309,-75.831,-176.685,8.652,148.753
C04351=1154.115,324.062,-75.800,-176.687,8.648,148.753
C04352=1154.120,323.814,-75.767,-176.689,8.645,148.753
C04353=1154.123,323.566,-75.735,-176.692,8.641,148.753
C04354=1154.128,323.318,-75.702,-176.695,8.638,148.752
C04355=1154.131,323.070,-75.670,-176.697,8.634,148.752
C04356=1154.136,322.822,-75.637,-176.700,8.631,148.752
C04357=1154.140,322.575,-75.606,-176.703,8.627,148.752
C04358=1154.144,322.326,-75.573,-176.705,8.624,148.752
C04359=1154.148,322.079,-75.541,-176.707,8.621,148.752
C04360=1154.152,321.831,-75.508,-176.710,8.617,148.751
C04361=1154.156,321.583,-75.476,-176.712,8.613,148.751
C04362=1154.161,321.335,-75.444,-176.715,8.610,148.751
C04363=1154.164,321.088,-75.412,-176.718,8.606,148.751
C04364=1154.169,320.839,-75.379,-176.720,8.603,148.751
C04365=1154.172,320.591,-75.348,-176.723,8.600,148.751
C04366=1154.177,320.343,-75.315,-176.725,8.597,148.750
C04367=1154.181,320.095,-75.284,-176.728,8.593,148.750
C04368=1154.185,319.847,-75.252,-176.731,8.589,148.750
C04369=1154.189,319.599,-75.219,-176.733,8.586,148.750
C04370=1154.193,319.352,-75.187,-176.736,8.582,148.750
C04371=1154.197,319.104,-75.155,-176.738,8.579,148.750
C04372=1154.201,318.856,-75.123,-176.741,8.576,148.750
C04373=1154.205,318.608,-75.091,-176.743,8.573,148.749
C04374=1154.210,318.360,-75.059,-176.746,8.569,148.749
C04375=1154.214,318.112,-75.027,-176.748,8.565,148.749
C04376=1154.218,317.864,-74.995,-176.751,8.562,148.749
C04377=1154.223,317.617,-74.963,-176.754,8.558,148.749
C04378=1154.226,317.368,-74.931,-176.756,8.555,148.749
C04379=1154.230,317.120,-74.899,-176.759,8.552,148.748
C04380=1154.234,316.873,-74.868,-176.761,8.548,148.748
C04381=1154.239,316.625,-74.836,-176.764,8.545,148.748
C04382=1154.243,316.377,-74.804,-176.767,8.541,148.748
C04383=1154.247,316.129,-74.772,-176.769,8.538,148.748
C04384=1154.251,315.881,-74.740,-176.771,8.535,148.748
C04385=1154.255,315.632,-74.709,-176.775,8.531,148.748
C04386=1154.260,315.385,-74.677,-176.777,8.528,148.747
C04387=1154.263,315.137,-74.645,-176.779,8.524,148.747
C04388=1154.268,314.889,-74.613,-176.782,8.521,148.747
C04389=1154.272,314.641,-74.581,-176.785,8.517,148.747
C04390=1154.276,314.393,-74.550,-176.787,8.514,148.747
C04391=1154.280,314.146,-74.518,-176.790,8.511,148.747
C04392=1154.285,313.868,-74.483,-176.792,8.507,148.746
C04393=1154.289,313.590,-74.448,-176.796,8.503,148.746
C04394=1154.294,313.313,-74.412,-176.799,8.499,148.746
C04395=1154.299,313.036,-74.376,-176.801,8.496,148.746
C04396=1154.303,312.788,-74.344,-176.804,8.493,148.746
C04397=1154.307,312.540,-74.314,-176.807,8.489,148.746
C04398=1154.311,312.292,-74.282,-176.809,8.485,148.746
C04399=1154.315,312.044,-74.250,-176.812,8.482,148.746
C04400=1154.319,311.796,-74.219,-176.814,8.479,148.745
C04401=1154.323,311.548,-74.187,-176.817,8.475,148.745
C04402=1154.327,311.300,-74.156,-176.819,8.472,148.745
C04403=1154.332,311.051,-74.124,-176.822,8.469,148.745
C04404=1154.336,310.804,-74.093,-176.824,8.465,148.745
C04405=1154.340,310.555,-74.061,-176.827,8.461,148.745
C04406=1154.345,310.308,-74.030,-176.830,8.458,148.745
C04407=1154.348,310.060,-73.998,-176.832,8.455,148.744
C04408=1154.353,309.812,-73.967,-176.835,8.452,148.744
C04409=1154.357,309.564,-73.935,-176.838,8.448,148.744
C04410=1154.361,309.316,-73.905,-176.840,8.445,148.744
C04411=1154.365,309.068,-73.873,-176.843,8.441,148.744
C04412=1154.370,308.820,-73.842,-176.845,8.439,148.744
C04413=1154.373,308.572,-73.810,-176.848,8.435,148.744
C04414=1154.378,308.324,-73.780,-176.851,8.431,148.744
C04415=1154.382,308.076,-73.748,-176.853,8.428,148.744
C04416=1154.386,307.828,-73.717,-176.856,8.425,148.743
C04417=1154.390,307.580,-73.685,-176.858,8.422,148.743
C04418=1154.395,307.332,-73.654,-176.861,8.418,148.743
C04419=1154.399,307.083,-73.623,-176.864,8.415,148.743
C04420=1154.403,306.836,-73.592,-176.866,8.412,148.743
C04421=1154.408,306.588,-73.561,-176.869,8.408,148.743
C04422=1154.411,306.340,-73.529,-176.871,8.405,148.743
C04423=1154.416,306.092,-73.498,-176.874,8.401,148.743
C04424=1154.420,305.843,-73.467,-176.877,8.398,148.742
C04425=1154.424,305.596,-73.436,-176.879,8.395,148.742
C04426=1154.428,305.348,-73.405,-176.882,8.392,148.742
C04427=1154.432,305.100,-73.374,-176.884,8.389,148.742
C04428=1154.436,304.852,-73.343,-176.887,8.385,148.742
C04429=1154.440,304.604,-73.312,-176.890,8.381,148.742
C04430=1154.445,304.356,-73.281,-176.892,8.378,148.742
C04431=1154.449,304.107,-73.250,-176.895,8.375,148.742
C04432=1154.454,303.859,-73.219,-176.897,8.372,148.742
C04433=1154.458,303.612,-73.188,-176.900,8.368,148.742
C04434=1154.461,303.363,-73.157,-176.903,8.365,148.741
C04435=1154.466,303.115,-73.126,-176.905,8.362,148.741
C04436=1154.471,302.867,-73.096,-176.908,8.359,148.741
C04437=1154.475,302.619,-73.064,-176.910,8.355,148.741
C04438=1154.479,302.371,-73.033,-176.913,8.352,148.741
C04439=1154.483,302.124,-73.003,-176.916,8.348,148.741
C04440=1154.487,301.875,-72.972,-176.919,8.345,148.741
C04441=1154.491,301.627,-72.941,-176.921,8.342,148.741
C04442=1154.496,301.379,-72.910,-176.924,8.339,148.741
C04443=1154.499,301.131,-72.880,-176.926,8.336,148.741
C04444=1154.504,300.883,-72.849,-176.929,8.333,148.741
C04445=1154.508,300.635,-72.818,-176.932,8.329,148.740
C04446=1154.512,300.386,-72.787,-176.934,8.326,148.740
C04447=1154.516,300.139,-72.757,-176.937,8.323,148.740
C04448=1154.521,299.891,-72.726,-176.939,8.319,148.740
C04449=1154.525,299.642,-72.695,-176.942,8.316,148.740
C04450=1154.529,299.394,-72.665,-176.944,8.313,148.740
C04451=1154.533,299.146,-72.634,-176.947,8.309,148.740
C04452=1154.537,298.898,-72.603,-176.950,8.306,148.740
C04453=1154.541,298.650,-72.573,-176.952,8.303,148.740
C04454=1154.546,298.402,-72.542,-176.955,8.300,148.740
C04455=1154.551,298.154,-72.511,-176.958,8.297,148.740
C04456=1154.554,297.906,-72.481,-176.960,8.294,148.739
C04457=1154.558,297.658,-72.450,-176.963,8.290,148.739
C04458=1154.563,297.410,-72.419,-176.965,8.287,148.739
C04459=1154.567,297.162,-72.390,-176.968,8.284,148.739
C04460=1154.571,296.913,-72.358,-176.971,8.280,148.739
C04461=1154.575,296.665,-72.328,-176.973,8.277,148.739
C04462=1154.580,296.417,-72.298,-176.976,8.274,148.739
C04463=1154.584,296.170,-72.267,-176.978,8.271,148.739
C04464=1154.588,295.921,-72.237,-176.981,8.267,148.739
C04465=1154.593,295.673,-72.206,-176.984,8.264,148.739
C04466=1154.596,295.425,-72.176,-176.986,8.261,148.739
C04467=1154.601,295.177,-72.145,-176.989,8.258,148.739
C04468=1154.605,294.929,-72.116,-176.991,8.255,148.738
C04469=1154.609,294.680,-72.085,-176.994,8.252,148.739
C04470=1154.613,294.432,-72.055,-176.997,8.248,148.738
C04471=1154.618,294.184,-72.024,-177.000,8.245,148.738
C04472=1154.622,293.936,-71.994,-177.002,8.241,148.738
C04473=1154.627,293.688,-71.964,-177.005,8.238,148.738
C04474=1154.630,293.441,-71.933,-177.008,8.235,148.738
C04475=1154.634,293.192,-71.904,-177.010,8.232,148.738
C04476=1154.639,292.944,-71.873,-177.013,8.229,148.738
C04477=1154.643,292.695,-71.843,-177.015,8.226,148.738
C04478=1154.647,292.447,-71.813,-177.018,8.223,148.738
C04479=1154.651,292.200,-71.782,-177.021,8.219,148.738
C04480=1154.656,291.951,-71.752,-177.024,8.216,148.738
C04481=1154.659,291.703,-71.722,-177.026,8.213,148.738
C04482=1154.664,291.455,-71.692,-177.029,8.210,148.738
C04483=1154.668,291.207,-71.662,-177.031,8.207,148.738
C04484=1154.672,290.958,-71.632,-177.034,8.203,148.738
C04485=1154.677,290.710,-71.601,-177.036,8.200,148.738
C04486=1154.681,290.462,-71.572,-177.039,8.197,148.737
C04487=1154.685,290.214,-71.542,-177.042,8.193,148.737
C04488=1154.690,289.966,-71.512,-177.045,8.190,148.737
C04489=1154.694,289.718,-71.482,-177.047,8.187,148.737
C04490=1154.698,289.470,-71.452,-177.050,8.184,148.737
C04491=1154.702,289.221,-71.422,-177.052,8.181,148.737
C04492=1154.706,288.973,-71.392,-177.055,8.178,148.737
C04493=1154.710,288.725,-71.362,-177.058,8.175,148.737
C04494=1154.714,288.477,-71.332,-177.060,8.172,148.737
C04495=1154.719,288.229,-71.302,-177.063,8.169,148.737
C04496=1154.724,287.954,-71.269,-177.066,8.165,148.737
C04497=1154.729,287.678,-71.236,-177.069,8.162,148.737
C04498=1154.733,287.404,-71.203,-177.072,8.158,148.737
C04499=1154.738,287.128,-71.170,-177.075,8.154,148.737
C04500=1154.742,286.879,-71.140,-177.078,8.151,148.737
C04501=1154.746,286.632,-71.110,-177.080,8.148,148.737
C04502=1154.751,286.383,-71.080,-177.083,8.145,148.737
C04503=1154.755,286.135,-71.051,-177.085,8.142,148.737
C04504=1154.759,285.887,-71.021,-177.088,8.139,148.737
C04505=1154.763,285.639,-70.991,-177.090,8.136,148.736
C04506=1154.767,285.391,-70.961,-177.093,8.133,148.737
C04507=1154.772,285.142,-70.931,-177.096,8.130,148.737
C04508=1154.776,284.894,-70.902,-177.098,8.126,148.736
C04509=1154.781,284.646,-70.873,-177.101,8.123,148.736
C04510=1154.785,284.399,-70.843,-177.104,8.121,148.736
C04511=1154.789,284.150,-70.813,-177.106,8.117,148.736
C04512=1154.793,283.902,-70.784,-177.109,8.113,148.736
C04513=1154.798,283.653,-70.754,-177.112,8.111,148.736
C04514=1154.802,283.405,-70.724,-177.115,8.107,148.736
C04515=1154.807,283.157,-70.695,-177.117,8.104,148.736
C04516=1154.811,282.909,-70.665,-177.120,8.101,148.736
C04517=1154.815,282.660,-70.636,-177.122,8.098,148.736
C04518=1154.819,282.412,-70.606,-177.125,8.095,148.736
C04519=1154.823,282.164,-70.577,-177.128,8.092,148.736
C04520=1154.828,281.916,-70.548,-177.131,8.089,148.736
C04521=1154.832,281.667,-70.518,-177.133,8.086,148.736
C04522=1154.836,281.419,-70.489,-177.136,8.083,148.736
C04523=1154.840,281.171,-70.459,-177.139,8.080,148.736
C04524=1154.845,280.923,-70.430,-177.141,8.077,148.736
C04525=1154.849,280.675,-70.401,-177.144,8.074,148.736
C04526=1154.853,280.427,-70.371,-177.146,8.071,148.736
C04527=1154.857,280.178,-70.342,-177.149,8.068,148.736
C04528=1154.862,279.930,-70.312,-177.152,8.064,148.736
C04529=1154.866,279.682,-70.283,-177.155,8.061,148.736
C04530=1154.870,279.434,-70.253,-177.158,8.058,148.736
C04531=1154.874,279.185,-70.225,-177.160,8.055,148.736
C04532=1154.879,278.937,-70.196,-177.163,8.052,148.736
C04533=1154.883,278.689,-70.166,-177.165,8.049,148.736
C04534=1154.888,278.441,-70.137,-177.168,8.046,148.736
C04535=1154.892,278.192,-70.107,-177.170,8.043,148.736
C04536=1154.896,277.944,-70.078,-177.173,8.040,148.736
C04537=1154.900,277.695,-70.049,-177.176,8.037,148.736
C04538=1154.905,277.448,-70.020,-177.179,8.034,148.736
C04539=1154.909,277.199,-69.990,-177.181,8.030,148.736
C04540=1154.914,276.951,-69.961,-177.184,8.027,148.736
C04541=1154.917,276.703,-69.933,-177.187,8.025,148.736
C04542=1154.921,276.454,-69.903,-177.189,8.022,148.736
C04543=1154.926,276.207,-69.874,-177.192,8.018,148.736
C04544=1154.931,275.958,-69.846,-177.194,8.015,148.736
C04545=1154.935,275.710,-69.816,-177.197,8.012,148.736
C04546=1154.939,275.461,-69.787,-177.200,8.009,148.736
C04547=1154.943,275.213,-69.759,-177.202,8.006,148.736
C04548=1154.948,274.965,-69.729,-177.205,8.003,148.736
C04549=1154.952,274.717,-69.700,-177.208,8.000,148.736
C04550=1154.956,274.468,-69.671,-177.211,7.997,148.736
C04551=1154.961,274.220,-69.642,-177.213,7.994,148.736
C04552=1154.965,273.972,-69.614,-177.216,7.991,148.736
C04553=1154.969,273.724,-69.585,-177.218,7.988,148.736
C04554=1154.974,273.475,-69.556,-177.221,7.985,148.736
C04555=1154.978,273.226,-69.526,-177.224,7.982,148.736
C04556=1154.982,272.979,-69.498,-177.227,7.979,148.736
C04557=1154.986,272.730,-69.469,-177.229,7.976,148.736
C04558=1154.990,272.482,-69.440,-177.232,7.973,148.736
C04559=1154.995,272.233,-69.411,-177.235,7.970,148.736
C04560=1154.999,271.985,-69.383,-177.237,7.967,148.736
C04561=1155.003,271.737,-69.354,-177.240,7.964,148.736
C04562=1155.008,271.488,-69.325,-177.242,7.961,148.736
C04563=1155.012,271.241,-69.297,-177.245,7.958,148.736
C04564=1155.016,270.992,-69.268,-177.248,7.955,148.736
C04565=1155.021,270.744,-69.238,-177.251,7.952,148.736
C04566=1155.025,270.496,-69.211,-177.254,7.949,148.736
C04567=1155.029,270.247,-69.182,-177.256,7.946,148.736
C04568=1155.034,269.999,-69.152,-177.259,7.943,148.736
C04569=1155.038,269.751,-69.125,-177.261,7.940,148.736
C04570=1155.043,269.502,-69.096,-177.264,7.937,148.736
C04571=1155.047,269.254,-69.066,-177.267,7.934,148.736
C04572=1155.051,269.006,-69.039,-177.270,7.931,148.736
C04573=1155.056,268.757,-69.010,-177.272,7.928,148.736
C04574=1155.060,268.510,-68.981,-177.275,7.925,148.736
C04575=1155.064,268.261,-68.953,-177.278,7.922,148.736
C04576=1155.069,268.012,-68.924,-177.280,7.919,148.736
C04577=1155.073,267.764,-68.896,-177.283,7.916,148.736
C04578=1155.077,267.516,-68.867,-177.286,7.913,148.736
C04579=1155.081,267.267,-68.839,-177.289,7.910,148.736
C04580=1155.086,267.019,-68.810,-177.291,7.907,148.736
C04581=1155.090,266.770,-68.782,-177.294,7.904,148.737
C04582=1155.095,266.522,-68.754,-177.297,7.901,148.736
C04583=1155.099,266.274,-68.725,-177.299,7.898,148.736
C04584=1155.103,266.026,-68.696,-177.302,7.895,148.736
C04585=1155.107,265.777,-68.668,-177.305,7.892,148.737
C04586=1155.112,265.529,-68.640,-177.308,7.889,148.737
C04587=1155.116,265.281,-68.612,-177.310,7.886,148.737
C04588=1155.120,265.032,-68.583,-177.313,7.883,148.737
C04589=1155.125,264.784,-68.555,-177.316,7.881,148.737
C04590=1155.129,264.535,-68.526,-177.319,7.878,148.737
C04591=1155.134,264.287,-68.499,-177.321,7.874,148.737
C04592=1155.138,264.038,-68.470,-177.324,7.871,148.737
C04593=1155.142,263.790,-68.442,-177.326,7.869,148.737
C04594=1155.147,263.541,-68.413,-177.329,7.866,148.737
C04595=1155.151,263.294,-68.386,-177.331,7.863,148.737
C04596=1155.155,263.045,-68.358,-177.334,7.860,148.737
C04597=1155.160,262.797,-68.329,-177.337,7.857,148.737
C04598=1155.164,262.548,-68.301,-177.340,7.855,148.737
C04599=1155.169,262.300,-68.273,-177.343,7.852,148.737
C04600=1155.174,262.027,-68.242,-177.346,7.848,148.737
C04601=1155.178,261.753,-68.211,-177.349,7.845,148.737
C04602=1155.183,261.481,-68.180,-177.351,7.842,148.737
C04603=1155.187,261.207,-68.149,-177.354,7.839,148.737
C04604=1155.192,260.958,-68.120,-177.357,7.836,148.737
C04605=1155.196,260.710,-68.093,-177.360,7.833,148.737
C04606=1155.200,260.461,-68.065,-177.363,7.830,148.738
C04607=1155.205,260.213,-68.037,-177.365,7.827,148.738
C04608=1155.209,259.965,-68.009,-177.368,7.824,148.738
C04609=1155.213,259.717,-67.981,-177.371,7.821,148.738
C04610=1155.217,259.468,-67.954,-177.374,7.818,148.738
C04611=1155.222,259.219,-67.925,-177.376,7.815,148.738
C04612=1155.227,258.972,-67.897,-177.379,7.812,148.738
C04613=1155.231,258.723,-67.869,-177.381,7.809,148.738
C04614=1155.235,258.475,-67.842,-177.384,7.806,148.738
C04615=1155.240,258.226,-67.813,-177.387,7.803,148.738
C04616=1155.244,257.978,-67.786,-177.390,7.800,148.738
C04617=1155.248,257.730,-67.758,-177.392,7.798,148.738
C04618=1155.252,257.481,-67.730,-177.395,7.795,148.738
C04619=1155.258,257.232,-67.702,-177.398,7.792,148.738
C04620=1155.261,256.984,-67.674,-177.400,7.789,148.738
C04621=1155.266,256.735,-67.647,-177.403,7.787,148.738
C04622=1155.270,256.487,-67.619,-177.406,7.784,148.738
C04623=1155.274,256.239,-67.591,-177.409,7.781,148.738
C04624=1155.279,255.990,-67.564,-177.411,7.778,148.738
C04625=1155.284,255.742,-67.536,-177.414,7.775,148.739
C04626=1155.288,255.493,-67.508,-177.417,7.772,148.739
C04627=1155.292,255.245,-67.480,-177.419,7.770,148.739
C04628=1155.297,254.997,-67.453,-177.422,7.767,148.739
C04629=1155.301,254.748,-67.425,-177.425,7.764,148.739
C04630=1155.305,254.500,-67.398,-177.427,7.761,148.739
C04631=1155.310,254.252,-67.370,-177.430,7.758,148.739
C04632=1155.314,254.002,-67.343,-177.433,7.755,148.739
C04633=1155.318,253.755,-67.315,-177.436,7.752,148.739
C04634=1155.323,253.506,-67.288,-177.439,7.749,148.739
C04635=1155.326,253.258,-67.260,-177.441,7.746,148.739
C04636=1155.332,253.009,-67.232,-177.444,7.744,148.739
C04637=1155.336,252.761,-67.204,-177.446,7.741,148.739
C04638=1155.341,252.512,-67.177,-177.449,7.738,148.739
C04639=1155.345,252.264,-67.149,-177.452,7.735,148.739
C04640=1155.349,252.015,-67.122,-177.455,7.733,148.740
C04641=1155.354,251.767,-67.095,-177.458,7.730,148.740
C04642=1155.358,251.518,-67.067,-177.461,7.727,148.740
C04643=1155.362,251.270,-67.040,-177.463,7.724,148.740
C04644=1155.367,251.021,-67.013,-177.466,7.722,148.740
C04645=1155.371,250.773,-66.985,-177.468,7.719,148.740
C04646=1155.375,250.524,-66.958,-177.471,7.716,148.740
C04647=1155.379,250.276,-66.931,-177.474,7.713,148.740
C04648=1155.384,250.028,-66.903,-177.477,7.710,148.740
C04649=1155.388,249.780,-66.876,-177.479,7.707,148.740
C04650=1155.392,249.530,-66.849,-177.482,7.704,148.740
C04651=1155.397,249.282,-66.822,-177.485,7.701,148.741
C04652=1155.401,249.034,-66.794,-177.487,7.699,148.741
C04653=1155.406,248.786,-66.767,-177.490,7.696,148.741
C04654=1155.411,248.537,-66.740,-177.493,7.693,148.741
C04655=1155.415,248.288,-66.713,-177.496,7.690,148.741
C04656=1155.419,248.039,-66.686,-177.499,7.688,148.741
C04657=1155.424,247.791,-66.658,-177.502,7.685,148.741
C04658=1155.428,247.543,-66.631,-177.504,7.682,148.741
C04659=1155.432,247.295,-66.604,-177.507,7.680,148.741
C04660=1155.437,247.046,-66.577,-177.509,7.677,148.741
C04661=1155.441,246.797,-66.550,-177.512,7.674,148.742
C04662=1155.446,246.549,-66.523,-177.515,7.671,148.742
C04663=1155.450,246.300,-66.496,-177.518,7.668,148.742
C04664=1155.454,246.052,-66.469,-177.520,7.665,148.742
C04665=1155.459,245.803,-66.442,-177.523,7.663,148.742
C04666=1155.464,245.555,-66.415,-177.525,7.660,148.742
C04667=1155.468,245.306,-66.388,-177.529,7.657,148.742
C04668=1155.472,245.057,-66.361,-177.531,7.654,148.742
C04669=1155.476,244.809,-66.334,-177.534,7.651,148.742
C04670=1155.481,244.561,-66.307,-177.537,7.648,148.742
C04671=1155.486,244.312,-66.280,-177.539,7.646,148.743
C04672=1155.490,244.064,-66.253,-177.542,7.643,148.743
C04673=1155.494,243.815,-66.226,-177.545,7.640,148.743
C04674=1155.499,243.567,-66.199,-177.547,7.637,148.743
C04675=1155.503,243.318,-66.172,-177.551,7.635,148.743
C04676=1155.507,243.070,-66.146,-177.553,7.633,148.743
C04677=1155.512,242.822,-66.119,-177.556,7.630,148.743
C04678=1155.516,242.573,-66.091,-177.558,7.627,148.743
C04679=1155.520,242.324,-66.065,-177.561,7.624,148.743
C04680=1155.525,242.076,-66.038,-177.564,7.621,148.743
C04681=1155.529,241.827,-66.011,-177.566,7.619,148.744
C04682=1155.534,241.579,-65.985,-177.569,7.616,148.744
C04683=1155.538,241.330,-65.958,-177.572,7.613,148.744
C04684=1155.543,241.082,-65.931,-177.575,7.610,148.744
C04685=1155.547,240.833,-65.904,-177.578,7.607,148.744
C04686=1155.551,240.585,-65.877,-177.581,7.605,148.744
C04687=1155.556,240.336,-65.851,-177.583,7.602,148.744
C04688=1155.560,240.088,-65.825,-177.586,7.600,148.745
C04689=1155.565,239.839,-65.797,-177.589,7.597,148.745
C04690=1155.569,239.591,-65.771,-177.592,7.594,148.745
C04691=1155.574,239.342,-65.745,-177.594,7.592,148.745
C04692=1155.578,239.094,-65.718,-177.597,7.589,148.745
C04693=1155.582,238.845,-65.691,-177.599,7.586,148.745
C04694=1155.587,238.596,-65.665,-177.603,7.583,148.745
C04695=1155.591,238.348,-65.638,-177.605,7.580,148.745
C04696=1155.596,238.099,-65.611,-177.608,7.578,148.745
C04697=1155.600,237.850,-65.585,-177.610,7.575,148.745
C04698=1155.605,237.602,-65.558,-177.613,7.572,148.746
C04699=1155.609,237.354,-65.532,-177.616,7.570,148.746
C04700=1155.614,237.105,-65.506,-177.619,7.567,148.746
C04701=1155.618,236.857,-65.479,-177.621,7.565,148.746
C04702=1155.623,236.607,-65.453,-177.624,7.562,148.746
C04703=1155.627,236.359,-65.426,-177.627,7.559,148.746
C04704=1155.632,236.087,-65.398,-177.630,7.556,148.746
C04705=1155.636,235.816,-65.369,-177.633,7.553,148.747
C04706=1155.641,235.544,-65.340,-177.636,7.550,148.747
C04707=1155.646,235.272,-65.312,-177.639,7.548,148.747
C04708=1155.651,235.024,-65.284,-177.642,7.545,148.747
C04709=1155.655,234.775,-65.259,-177.644,7.542,148.747
C04710=1155.660,234.526,-65.232,-177.647,7.539,148.747
C04711=1155.664,234.278,-65.206,-177.649,7.537,148.747
C04712=1155.668,234.029,-65.179,-177.653,7.534,148.748
C04713=1155.673,233.781,-65.153,-177.655,7.531,148.748
C04714=1155.678,233.532,-65.128,-177.658,7.528,148.748
C04715=1155.682,233.284,-65.101,-177.660,7.526,148.748
C04716=1155.686,233.035,-65.075,-177.664,7.524,148.748
C04717=1155.690,232.787,-65.048,-177.666,7.521,148.748
C04718=1155.695,232.538,-65.022,-177.669,7.518,148.748
C04719=1155.700,232.289,-64.996,-177.671,7.516,148.748
C04720=1155.704,232.041,-64.970,-177.675,7.513,148.749
C04721=1155.709,231.792,-64.944,-177.677,7.510,148.749
C04722=1155.713,231.543,-64.918,-177.680,7.508,148.749
C04723=1155.717,231.295,-64.892,-177.682,7.505,148.749
C04724=1155.721,231.046,-64.866,-177.686,7.503,148.749
C04725=1155.726,230.797,-64.840,-177.688,7.500,148.749
C04726=1155.731,230.549,-64.814,-177.691,7.498,148.749
C04727=1155.735,230.301,-64.788,-177.693,7.495,148.750
C04728=1155.740,230.052,-64.761,-177.697,7.492,148.750
C04729=1155.744,229.803,-64.736,-177.699,7.489,148.750
C04730=1155.749,229.554,-64.710,-177.702,7.487,148.750
C04731=1155.753,229.307,-64.684,-177.704,7.484,148.750
C04732=1155.757,229.058,-64.658,-177.708,7.481,148.750
C04733=1155.762,228.809,-64.632,-177.710,7.479,148.751
C04734=1155.766,228.560,-64.606,-177.713,7.476,148.751
C04735=1155.771,228.311,-64.580,-177.716,7.474,148.751
C04736=1155.776,228.063,-64.555,-177.719,7.471,148.751
C04737=1155.780,227.814,-64.529,-177.721,7.469,148.751
C04738=1155.784,227.566,-64.502,-177.724,7.466,148.751
C04739=1155.789,227.317,-64.476,-177.727,7.463,148.752
C04740=1155.793,227.069,-64.451,-177.729,7.461,148.752
C04741=1155.798,226.820,-64.425,-177.732,7.458,148.752
C04742=1155.802,226.571,-64.399,-177.735,7.456,148.752
C04743=1155.806,226.323,-64.374,-177.737,7.453,148.752
C04744=1155.811,226.074,-64.348,-177.740,7.451,148.752
C04745=1155.816,225.825,-64.322,-177.743,7.448,148.752
C04746=1155.820,225.577,-64.296,-177.746,7.445,148.753
C04747=1155.825,225.328,-64.271,-177.748,7.443,148.753
C04748=1155.829,225.080,-64.245,-177.751,7.440,148.753
C04749=1155.833,224.831,-64.219,-177.754,7.437,148.753
C04750=1155.838,224.583,-64.194,-177.757,7.435,148.753
C04751=1155.842,224.334,-64.168,-177.759,7.432,148.753
C04752=1155.847,224.085,-64.142,-177.763,7.430,148.754
C04753=1155.851,223.836,-64.117,-177.765,7.428,148.754
C04754=1155.856,223.588,-64.092,-177.768,7.425,148.754
C04755=1155.860,223.339,-64.066,-177.771,7.422,148.754
C04756=1155.865,223.090,-64.040,-177.773,7.420,148.754
C04757=1155.869,222.842,-64.015,-177.776,7.417,148.754
C04758=1155.874,222.593,-63.989,-177.779,7.414,148.755
C04759=1155.878,222.345,-63.964,-177.781,7.412,148.755
C04760=1155.883,222.096,-63.938,-177.784,7.409,148.755
C04761=1155.887,221.847,-63.913,-177.787,7.407,148.755
C04762=1155.892,221.599,-63.888,-177.790,7.405,148.755
C04763=1155.896,221.350,-63.862,-177.792,7.402,148.755
C04764=1155.900,221.101,-63.836,-177.796,7.399,148.756
C04765=1155.906,220.852,-63.812,-177.798,7.397,148.756
C04766=1155.910,220.603,-63.786,-177.801,7.394,148.756
C04767=1155.915,220.355,-63.760,-177.804,7.392,148.756
C04768=1155.919,220.107,-63.735,-177.806,7.389,148.756
C04769=1155.923,219.857,-63.710,-177.809,7.387,148.756
C04770=1155.928,219.609,-63.684,-177.811,7.385,148.757
C04771=1155.932,219.360,-63.659,-177.814,7.382,148.757
C04772=1155.937,219.112,-63.634,-177.818,7.379,148.757
C04773=1155.941,218.863,-63.609,-177.820,7.377,148.757
C04774=1155.945,218.614,-63.583,-177.823,7.374,148.757
C04775=1155.950,218.365,-63.558,-177.826,7.372,148.758
C04776=1155.955,218.117,-63.533,-177.828,7.370,148.758
C04777=1155.959,217.869,-63.507,-177.831,7.367,148.758
C04778=1155.964,217.619,-63.482,-177.833,7.365,148.758
C04779=1155.968,217.371,-63.457,-177.836,7.362,148.758
C04780=1155.973,217.122,-63.432,-177.839,7.359,148.759
C04781=1155.977,216.874,-63.407,-177.842,7.357,148.759
C04782=1155.982,216.624,-63.382,-177.844,7.354,148.759
C04783=1155.987,216.376,-63.356,-177.848,7.352,148.759
C04784=1155.991,216.127,-63.332,-177.850,7.350,148.759
C04785=1155.995,215.879,-63.307,-177.853,7.347,148.759
C04786=1156.000,215.630,-63.282,-177.855,7.345,148.760
C04787=1156.005,215.382,-63.256,-177.858,7.342,148.760
C04788=1156.009,215.132,-63.232,-177.861,7.339,148.760
C04789=1156.013,214.884,-63.206,-177.864,7.337,148.760
C04790=1156.018,214.635,-63.181,-177.866,7.334,148.760
C04791=1156.023,214.387,-63.156,-177.869,7.333,148.761
C04792=1156.027,214.138,-63.132,-177.872,7.330,148.761
C04793=1156.031,213.890,-63.106,-177.875,7.327,148.761
C04794=1156.036,213.640,-63.081,-177.877,7.325,148.761
C04795=1156.040,213.392,-63.057,-177.881,7.322,148.762
C04796=1156.044,213.143,-63.031,-177.883,7.320,148.762
C04797=1156.050,212.894,-63.007,-177.886,7.317,148.762
C04798=1156.054,212.645,-62.982,-177.889,7.315,148.762
C04799=1156.058,212.397,-62.957,-177.891,7.313,148.762
C04800=1156.063,212.148,-62.932,-177.894,7.310,148.762
C04801=1156.067,211.899,-62.908,-177.896,7.308,148.763
C04802=1156.072,211.651,-62.882,-177.900,7.305,148.763
C04803=1156.077,211.402,-62.857,-177.902,7.303,148.763
C04804=1156.081,211.153,-62.833,-177.905,7.300,148.763
C04805=1156.085,210.904,-62.808,-177.908,7.298,148.763
C04806=1156.090,210.656,-62.783,-177.910,7.296,148.764
C04807=1156.095,210.407,-62.759,-177.913,7.293,148.764
C04808=1156.099,210.136,-62.732,-177.916,7.290,148.764
C04809=1156.104,209.866,-62.705,-177.919,7.288,148.764
C04810=1156.109,209.595,-62.678,-177.922,7.285,148.764
C04811=1156.114,209.325,-62.651,-177.925,7.283,148.765
C04812=1156.119,209.076,-62.626,-177.928,7.280,148.765
C04813=1156.123,208.827,-62.602,-177.930,7.278,148.765
C04814=1156.128,208.579,-62.577,-177.933,7.275,148.765
C04815=1156.133,208.329,-62.552,-177.936,7.273,148.766
C04816=1156.137,208.081,-62.528,-177.939,7.271,148.766
C04817=1156.142,207.832,-62.504,-177.941,7.269,148.766
C04818=1156.146,207.584,-62.478,-177.944,7.266,148.766
C04819=1156.151,207.335,-62.454,-177.947,7.263,148.766
C04820=1156.155,207.086,-62.430,-177.950,7.261,148.767
C04821=1156.160,206.837,-62.405,-177.953,7.259,148.767
C04822=1156.164,206.589,-62.381,-177.955,7.256,148.767
C04823=1156.169,206.340,-62.356,-177.958,7.254,148.767
C04824=1156.174,206.091,-62.332,-177.961,7.252,148.768
C04825=1156.177,205.842,-62.307,-177.964,7.249,148.768
C04826=1156.183,205.594,-62.283,-177.966,7.247,148.768
C04827=1156.187,205.345,-62.259,-177.969,7.244,148.768
C04828=1156.192,205.096,-62.234,-177.971,7.242,148.768
C04829=1156.196,204.847,-62.210,-177.975,7.240,148.769
C04830=1156.201,204.599,-62.185,-177.977,7.238,148.769
C04831=1156.205,204.350,-62.161,-177.980,7.235,148.769
C04832=1156.210,204.101,-62.137,-177.982,7.233,148.769
C04833=1156.215,203.852,-62.112,-177.986,7.230,148.770
C04834=1156.219,203.603,-62.088,-177.988,7.228,148.770
C04835=1156.223,203.355,-62.064,-177.991,7.226,148.770
C04836=1156.228,203.106,-62.039,-177.994,7.223,148.770
C04837=1156.232,202.857,-62.015,-177.997,7.221,148.771
C04838=1156.237,202.609,-61.991,-177.999,7.218,148.771
C04839=1156.242,202.360,-61.966,-178.002,7.216,148.771
C04840=1156.246,202.110,-61.943,-178.005,7.213,148.771
C04841=1156.250,201.862,-61.919,-178.008,7.212,148.771
C04842=1156.256,201.613,-61.894,-178.010,7.209,148.772
C04843=1156.260,201.365,-61.870,-178.013,7.207,148.772
C04844=1156.264,201.115,-61.846,-178.016,7.204,148.772
C04845=1156.269,200.866,-61.821,-178.018,7.202,148.772
C04846=1156.274,200.618,-61.797,-178.021,7.199,148.772
C04847=1156.278,200.369,-61.773,-178.024,7.198,148.773
C04848=1156.283,200.120,-61.750,-178.027,7.196,148.773
C04849=1156.288,199.872,-61.725,-178.029,7.193,148.773
C04850=1156.292,199.623,-61.701,-178.032,7.191,148.774
C04851=1156.296,199.374,-61.677,-178.035,7.188,148.774
C04852=1156.301,199.125,-61.653,-178.038,7.187,148.774
C04853=1156.305,198.877,-61.629,-178.040,7.184,148.774
C04854=1156.310,198.627,-61.605,-178.043,7.182,148.775
C04855=1156.315,198.379,-61.581,-178.046,7.179,148.775
C04856=1156.319,198.130,-61.557,-178.048,7.177,148.775
C04857=1156.323,197.881,-61.533,-178.051,7.174,148.775
C04858=1156.328,197.632,-61.509,-178.054,7.172,148.775
C04859=1156.333,197.384,-61.485,-178.057,7.170,148.776
C04860=1156.338,197.135,-61.461,-178.059,7.168,148.776
C04861=1156.342,196.886,-61.437,-178.063,7.165,148.776
C04862=1156.347,196.637,-61.414,-178.065,7.163,148.776
C04863=1156.351,196.389,-61.390,-178.068,7.161,148.777
C04864=1156.355,196.139,-61.366,-178.070,7.158,148.777
C04865=1156.360,195.891,-61.342,-178.074,7.156,148.777
C04866=1156.365,195.641,-61.318,-178.076,7.154,148.777
C04867=1156.369,195.393,-61.294,-178.079,7.152,148.778
C04868=1156.374,195.144,-61.271,-178.082,7.149,148.778
C04869=1156.379,194.895,-61.247,-178.084,7.147,148.778
C04870=1156.383,194.646,-61.223,-178.087,7.145,148.778
C04871=1156.388,194.398,-61.199,-178.090,7.143,148.779
C04872=1156.392,194.149,-61.176,-178.093,7.140,148.779
C04873=1156.397,193.900,-61.152,-178.095,7.138,148.779
C04874=1156.401,193.652,-61.128,-178.098,7.135,148.779
C04875=1156.406,193.402,-61.105,-178.101,7.134,148.780
C04876=1156.411,193.153,-61.082,-178.104,7.132,148.780
C04877=1156.415,192.905,-61.058,-178.106,7.129,148.780
C04878=1156.420,192.656,-61.034,-178.109,7.127,148.781
C04879=1156.424,192.408,-61.010,-178.112,7.124,148.781
C04880=1156.429,192.159,-60.987,-178.115,7.123,148.781
C04881=1156.434,191.910,-60.963,-178.118,7.120,148.781
C04882=1156.438,191.660,-60.940,-178.120,7.118,148.781
C04883=1156.443,191.412,-60.916,-178.123,7.116,148.782
C04884=1156.447,191.163,-60.893,-178.125,7.113,148.782
C04885=1156.452,190.914,-60.869,-178.128,7.111,148.782
C04886=1156.457,190.666,-60.845,-178.131,7.109,148.783
C04887=1156.461,190.417,-60.822,-178.134,7.107,148.783
C04888=1156.466,190.168,-60.798,-178.137,7.104,148.783
C04889=1156.471,189.919,-60.775,-178.140,7.102,148.783
C04890=1156.475,189.669,-60.752,-178.142,7.100,148.784
C04891=1156.480,189.421,-60.728,-178.145,7.098,148.784
C04892=1156.484,189.172,-60.704,-178.147,7.096,148.784
C04893=1156.489,188.923,-60.681,-178.151,7.093,148.784
C04894=1156.493,188.674,-60.658,-178.153,7.091,148.785
C04895=1156.498,188.425,-60.635,-178.155,7.089,148.785
C04896=1156.503,188.176,-60.612,-178.159,7.087,148.785
C04897=1156.507,187.927,-60.588,-178.161,7.085,148.786
C04898=1156.512,187.679,-60.564,-178.164,7.082,148.786
C04899=1156.516,187.430,-60.541,-178.167,7.080,148.786
C04900=1156.521,187.181,-60.517,-178.170,7.079,148.786
C04901=1156.525,186.932,-60.495,-178.172,7.076,148.786
C04902=1156.530,186.684,-60.472,-178.175,7.074,148.787
C04903=1156.535,186.435,-60.448,-178.178,7.072,148.787
C04904=1156.540,186.186,-60.425,-178.181,7.069,148.787
C04905=1156.544,185.937,-60.402,-178.183,7.067,148.788
C04906=1156.548,185.688,-60.379,-178.186,7.065,148.788
C04907=1156.553,185.439,-60.355,-178.189,7.063,148.788
C04908=1156.558,185.190,-60.332,-178.191,7.061,148.789
C04909=1156.562,184.941,-60.309,-178.195,7.058,148.789
C04910=1156.566,184.692,-60.286,-178.197,7.056,148.789
C04911=1156.572,184.444,-60.263,-178.200,7.054,148.789
C04912=1156.577,184.174,-60.238,-178.203,7.052,148.790
C04913=1156.582,183.903,-60.212,-178.206,7.049,148.790
C04914=1156.586,183.634,-60.188,-178.208,7.047,148.790
C04915=1156.591,183.365,-60.162,-178.212,7.045,148.791
C04916=1156.596,183.115,-60.140,-178.214,7.043,148.791
C04917=1156.601,182.867,-60.117,-178.218,7.040,148.791
C04918=1156.606,182.618,-60.094,-178.220,7.038,148.791
C04919=1156.610,182.369,-60.071,-178.223,7.036,148.792
C04920=1156.614,182.120,-60.048,-178.226,7.034,148.792
C04921=1156.619,181.871,-60.024,-178.228,7.032,148.792
C04922=1156.624,181.623,-60.001,-178.231,7.029,148.793
C04923=1156.629,181.374,-59.979,-178.234,7.028,148.793
C04924=1156.633,181.125,-59.956,-178.237,7.026,148.793
C04925=1156.638,180.876,-59.933,-178.239,7.023,148.793
C04926=1156.642,180.627,-59.910,-178.242,7.021,148.794
C04927=1156.648,180.378,-59.888,-178.245,7.019,148.794
C04928=1156.651,180.129,-59.865,-178.248,7.017,148.794
C04929=1156.656,179.880,-59.841,-178.250,7.015,148.795
C04930=1156.661,179.631,-59.818,-178.253,7.013,148.795
C04931=1156.666,179.383,-59.796,-178.256,7.011,148.795
C04932=1156.670,179.133,-59.773,-178.258,7.008,148.795
C04933=1156.674,178.885,-59.750,-178.261,7.007,148.796
C04934=1156.679,178.635,-59.728,-178.264,7.004,148.796
C04935=1156.684,178.387,-59.705,-178.267,7.002,148.796
C04936=1156.689,178.138,-59.682,-178.269,7.000,148.797
C04937=1156.693,177.889,-59.660,-178.273,6.998,148.797
C04938=1156.698,177.640,-59.637,-178.275,6.996,148.797
C04939=1156.703,177.391,-59.614,-178.277,6.994,148.797
C04940=1156.707,177.142,-59.591,-178.281,6.991,148.798
C04941=1156.712,176.893,-59.568,-178.283,6.990,148.798
C04942=1156.716,176.644,-59.546,-178.286,6.988,148.799
C04943=1156.721,176.395,-59.523,-178.288,6.986,148.799
C04944=1156.726,176.146,-59.501,-178.292,6.983,148.799
C04945=1156.730,175.897,-59.478,-178.294,6.981,148.799
C04946=1156.735,175.648,-59.456,-178.297,6.980,148.800
C04947=1156.739,175.400,-59.433,-178.300,6.977,148.800
C04948=1156.744,175.151,-59.410,-178.302,6.975,148.800
C04949=1156.749,174.902,-59.388,-178.305,6.973,148.801
C04950=1156.754,174.652,-59.366,-178.308,6.971,148.801
C04951=1156.758,174.404,-59.343,-178.311,6.969,148.801
C04952=1156.763,174.155,-59.320,-178.313,6.967,148.801
C04953=1156.767,173.906,-59.298,-178.316,6.965,148.802
C04954=1156.772,173.657,-59.276,-178.319,6.963,148.802
C04955=1156.777,173.408,-59.253,-178.322,6.961,148.803
C04956=1156.781,173.159,-59.231,-178.324,6.959,148.803
C04957=1156.786,172.911,-59.208,-178.328,6.956,148.803
C04958=1156.791,172.661,-59.186,-178.330,6.954,148.803
C04959=1156.795,172.412,-59.164,-178.333,6.953,148.804
C04960=1156.800,172.164,-59.141,-178.335,6.951,148.804
C04961=1156.805,171.914,-59.119,-178.338,6.948,148.804
C04962=1156.809,171.666,-59.097,-178.341,6.946,148.805
C04963=1156.814,171.416,-59.073,-178.344,6.944,148.805
C04964=1156.818,171.167,-59.051,-178.347,6.942,148.805
C04965=1156.823,170.919,-59.030,-178.349,6.940,148.806
C04966=1156.828,170.669,-59.006,-178.352,6.938,148.806
C04967=1156.833,170.421,-58.985,-178.355,6.936,148.806
C04968=1156.837,170.171,-58.963,-178.358,6.934,148.807
C04969=1156.841,169.922,-58.941,-178.361,6.932,148.807
C04970=1156.847,169.674,-58.918,-178.363,6.930,148.807
C04971=1156.851,169.424,-58.896,-178.366,6.928,148.807
C04972=1156.856,169.176,-58.874,-178.369,6.926,148.808
C04973=1156.861,168.926,-58.851,-178.372,6.924,148.808
C04974=1156.866,168.678,-58.830,-178.374,6.922,148.809
C04975=1156.870,168.429,-58.807,-178.376,6.920,148.809
C04976=1156.875,168.180,-58.785,-178.380,6.918,148.809
C04977=1156.879,167.931,-58.763,-178.382,6.916,148.809
C04978=1156.884,167.682,-58.741,-178.385,6.914,148.810
C04979=1156.889,167.433,-58.719,-178.388,6.912,148.810
C04980=1156.894,167.184,-58.697,-178.391,6.909,148.810
C04981=1156.898,166.935,-58.674,-178.393,6.908,148.811
C04982=1156.902,166.687,-58.653,-178.396,6.906,148.811
C04983=1156.907,166.437,-58.630,-178.399,6.904,148.811
C04984=1156.912,166.188,-58.608,-178.402,6.902,148.812
C04985=1156.917,165.939,-58.586,-178.405,6.900,148.812
C04986=1156.921,165.690,-58.565,-178.407,6.898,148.812
C04987=1156.926,165.441,-58.542,-178.410,6.896,148.813
C04988=1156.931,165.192,-58.521,-178.413,6.893,148.813
C04989=1156.935,164.943,-58.499,-178.416,6.892,148.813
C04990=1156.940,164.694,-58.476,-178.418,6.890,148.814
C04991=1156.945,164.445,-58.454,-178.421,6.888,148.814
C04992=1156.950,164.196,-58.433,-178.423,6.886,148.814
C04993=1156.954,163.947,-58.411,-178.426,6.884,148.815
C04994=1156.959,163.698,-58.389,-178.429,6.882,148.815
C04995=1156.963,163.449,-58.367,-178.432,6.880,148.815
C04996=1156.968,163.200,-58.345,-178.435,6.878,148.816
C04997=1156.973,162.951,-58.324,-178.437,6.877,148.816
C04998=1156.977,162.702,-58.302,-178.440,6.874,148.816
C04999=1156.982,162.453,-58.280,-178.443,6.872,148.817
C05000=1156.986,162.204,-58.258,-178.445,6.870,148.817
C05001=1156.991,161.955,-58.237,-178.448,6.869,148.817
C05002=1156.996,161.706,-58.215,-178.451,6.867,148.818
C05003=1157.000,161.457,-58.193,-178.454,6.864,148.818
C05004=1157.005,161.208,-58.171,-178.457,6.863,148.819
C05005=1157.010,160.959,-58.149,-178.459,6.861,148.819
C05006=1157.014,160.710,-58.128,-178.462,6.859,148.819
C05007=1157.020,160.461,-58.107,-178.464,6.857,148.819
C05008=1157.024,160.212,-58.085,-178.468,6.854,148.820
C05009=1157.029,159.963,-58.063,-178.470,6.853,148.820
C05010=1157.033,159.714,-58.041,-178.473,6.851,148.821
C05011=1157.038,159.465,-58.019,-178.476,6.849,148.821
C05012=1157.043,159.216,-57.998,-178.478,6.847,148.821
C05013=1157.047,158.966,-57.976,-178.482,6.845,148.822
C05014=1157.052,158.718,-57.955,-178.484,6.843,148.822
C05015=1157.057,158.469,-57.933,-178.487,6.841,148.822
C05016=1157.062,158.200,-57.910,-178.489,6.839,148.823
C05017=1157.067,157.931,-57.887,-178.493,6.837,148.823
C05018=1157.072,157.662,-57.864,-178.495,6.835,148.823
C05019=1157.077,157.393,-57.840,-178.499,6.833,148.824
C05020=1157.082,157.144,-57.819,-178.501,6.831,148.824
C05021=1157.087,156.894,-57.797,-178.504,6.829,148.824
C05022=1157.091,156.646,-57.776,-178.507,6.827,148.825
C05023=1157.096,156.397,-57.755,-178.509,6.826,148.825
C05024=1157.101,156.148,-57.733,-178.512,6.824,148.826
C05025=1157.105,155.899,-57.711,-178.515,6.821,148.826
C05026=1157.110,155.650,-57.690,-178.518,6.820,148.826
C05027=1157.115,155.401,-57.669,-178.521,6.818,148.827
C05028=1157.120,155.151,-57.647,-178.524,6.816,148.827
C05029=1157.124,154.903,-57.626,-178.526,6.814,148.827
C05030=1157.129,154.653,-57.605,-178.528,6.812,148.828
C05031=1157.134,154.405,-57.583,-178.531,6.811,148.828
C05032=1157.138,154.155,-57.562,-178.534,6.808,148.828
C05033=1157.143,153.906,-57.540,-178.537,6.806,148.829
C05034=1157.148,153.657,-57.520,-178.540,6.805,148.829
C05035=1157.153,153.408,-57.498,-178.543,6.803,148.829
C05036=1157.157,153.159,-57.477,-178.545,6.801,148.830
C05037=1157.162,152.910,-57.455,-178.548,6.799,148.830
C05038=1157.167,152.661,-57.435,-178.551,6.798,148.831
C05039=1157.171,152.412,-57.413,-178.554,6.795,148.831
C05040=1157.177,152.163,-57.392,-178.557,6.793,148.831
C05041=1157.181,151.914,-57.370,-178.559,6.792,148.832
C05042=1157.185,151.665,-57.350,-178.562,6.790,148.832
C05043=1157.190,151.415,-57.329,-178.565,6.788,148.832
C05044=1157.195,151.167,-57.307,-178.567,6.786,148.833
C05045=1157.200,150.918,-57.287,-178.570,6.784,148.833
C05046=1157.204,150.669,-57.265,-178.572,6.783,148.833
C05047=1157.209,150.419,-57.244,-178.576,6.780,148.834
C05048=1157.214,150.170,-57.224,-178.578,6.778,148.834
C05049=1157.219,149.922,-57.202,-178.581,6.777,148.835
C05050=1157.224,149.672,-57.181,-178.584,6.775,148.835
C05051=1157.228,149.424,-57.160,-178.586,6.773,148.835
C05052=1157.233,149.174,-57.139,-178.589,6.771,148.836
C05053=1157.238,148.925,-57.117,-178.592,6.770,148.836
C05054=1157.242,148.676,-57.097,-178.595,6.768,148.836
C05055=1157.247,148.427,-57.076,-178.597,6.766,148.837
C05056=1157.251,148.178,-57.055,-178.601,6.764,148.837
C05057=1157.256,147.929,-57.034,-178.603,6.762,148.838
C05058=1157.262,147.680,-57.013,-178.606,6.760,148.838
C05059=1157.266,147.431,-56.993,-178.609,6.758,148.838
C05060=1157.271,147.181,-56.971,-178.611,6.757,148.839
C05061=1157.275,146.933,-56.950,-178.614,6.755,148.839
C05062=1157.280,146.683,-56.929,-178.617,6.753,148.839
C05063=1157.284,146.434,-56.909,-178.619,6.752,148.840
C05064=1157.290,146.185,-56.888,-178.622,6.750,148.840
C05065=1157.295,145.936,-56.867,-178.625,6.748,148.841
C05066=1157.299,145.687,-56.847,-178.628,6.746,148.841
C05067=1157.304,145.438,-56.825,-178.631,6.744,148.841
C05068=1157.309,145.189,-56.805,-178.634,6.742,148.842
C05069=1157.314,144.940,-56.784,-178.636,6.740,148.842
C05070=1157.318,144.691,-56.763,-178.639,6.739,148.843
C05071=1157.323,144.442,-56.742,-178.642,6.737,148.843
C05072=1157.327,144.192,-56.722,-178.644,6.735,148.843
C05073=1157.332,143.943,-56.701,-178.647,6.733,148.843
C05074=1157.337,143.694,-56.680,-178.649,6.731,148.844
C05075=1157.341,143.445,-56.660,-178.652,6.730,148.844
C05076=1157.346,143.196,-56.639,-178.655,6.728,148.845
C05077=1157.351,142.947,-56.619,-178.657,6.726,148.845
C05078=1157.356,142.698,-56.598,-178.660,6.724,148.845
C05079=1157.360,142.449,-56.577,-178.663,6.723,148.846
C05080=1157.366,142.199,-56.556,-178.666,6.721,148.846
C05081=1157.370,141.950,-56.536,-178.668,6.719,148.847
C05082=1157.374,141.701,-56.515,-178.671,6.718,148.847
C05083=1157.380,141.452,-56.495,-178.675,6.715,148.848
C05084=1157.384,141.203,-56.474,-178.677,6.714,148.848
C05085=1157.389,140.954,-56.453,-178.680,6.712,148.848
C05086=1157.394,140.705,-56.433,-178.683,6.710,148.849
C05087=1157.398,140.456,-56.412,-178.686,6.708,148.849
C05088=1157.403,140.207,-56.391,-178.688,6.707,148.849
C05089=1157.408,139.957,-56.372,-178.691,6.705,148.850
C05090=1157.412,139.708,-56.351,-178.694,6.703,148.850
C05091=1157.418,139.459,-56.330,-178.696,6.702,148.851
C05092=1157.422,139.210,-56.310,-178.699,6.700,148.851
C05093=1157.427,138.961,-56.290,-178.702,6.698,148.851
C05094=1157.432,138.712,-56.269,-178.705,6.696,148.852
C05095=1157.436,138.462,-56.249,-178.707,6.695,148.852
C05096=1157.441,138.213,-56.229,-178.710,6.693,148.853
C05097=1157.446,137.965,-56.209,-178.713,6.691,148.853
C05098=1157.451,137.716,-56.188,-178.715,6.689,148.853
C05099=1157.456,137.467,-56.167,-178.718,6.688,148.854
C05100=1157.460,137.217,-56.148,-178.721,6.686,148.854
C05101=1157.465,136.968,-56.127,-178.724,6.684,148.855
C05102=1157.470,136.719,-56.106,-178.726,6.683,148.855
C05103=1157.474,136.470,-56.086,-178.729,6.681,148.855
C05104=1157.479,136.221,-56.066,-178.732,6.679,148.856
C05105=1157.484,135.971,-56.045,-178.734,6.677,148.856
C05106=1157.489,135.722,-56.025,-178.737,6.676,148.856
C05107=1157.493,135.473,-56.005,-178.740,6.674,148.857
C05108=1157.498,135.225,-55.985,-178.742,6.672,148.857
C05109=1157.503,134.976,-55.965,-178.745,6.671,148.858
C05110=1157.508,134.726,-55.945,-178.748,6.669,148.858
C05111=1157.513,134.477,-55.924,-178.751,6.667,148.858
C05112=1157.517,134.228,-55.904,-178.753,6.665,148.859
C05113=1157.522,133.978,-55.884,-178.756,6.664,148.859
C05114=1157.526,133.729,-55.864,-178.759,6.662,148.860
C05115=1157.532,133.481,-55.845,-178.762,6.661,148.860
C05116=1157.537,133.231,-55.824,-178.765,6.659,148.861
C05117=1157.541,132.982,-55.803,-178.767,6.657,148.861
C05118=1157.546,132.733,-55.784,-178.770,6.655,148.861
C05119=1157.551,132.484,-55.763,-178.773,6.654,148.862
C05120=1157.555,132.215,-55.742,-178.775,6.652,148.862
C05121=1157.561,131.946,-55.721,-178.778,6.650,148.863
C05122=1157.566,131.678,-55.699,-178.782,6.648,148.863
C05123=1157.571,131.409,-55.677,-178.785,6.646,148.864
C05124=1157.576,131.160,-55.657,-178.787,6.645,148.864
C05125=1157.581,130.911,-55.637,-178.790,6.643,148.864
C05126=1157.586,130.662,-55.618,-178.793,6.641,148.865
C05127=1157.590,130.413,-55.597,-178.796,6.639,148.865
C05128=1157.595,130.163,-55.578,-178.798,6.638,148.866
C05129=1157.600,129.915,-55.558,-178.801,6.636,148.866
C05130=1157.605,129.665,-55.538,-178.804,6.634,148.866
C05131=1157.609,129.417,-55.518,-178.807,6.633,148.867
C05132=1157.614,129.167,-55.498,-178.810,6.631,148.867
C05133=1157.619,128.918,-55.479,-178.812,6.630,148.868
C05134=1157.624,128.669,-55.458,-178.815,6.628,148.868
C05135=1157.629,128.420,-55.439,-178.817,6.627,148.869
C05136=1157.633,128.170,-55.419,-178.820,6.625,148.869
C05137=1157.638,127.922,-55.399,-178.823,6.623,148.869
C05138=1157.643,127.672,-55.379,-178.825,6.622,148.870
C05139=1157.648,127.423,-55.360,-178.828,6.620,148.870
C05140=1157.652,127.174,-55.339,-178.831,6.618,148.871
C05141=1157.658,126.925,-55.320,-178.834,6.617,148.871
C05142=1157.662,126.675,-55.300,-178.837,6.615,148.872
C05143=1157.667,126.426,-55.280,-178.839,6.614,148.872
C05144=1157.672,126.177,-55.260,-178.842,6.612,148.872
C05145=1157.677,125.928,-55.241,-178.845,6.610,148.873
C05146=1157.682,125.678,-55.221,-178.847,6.608,148.873
C05147=1157.686,125.429,-55.201,-178.850,6.607,148.874
C05148=1157.691,125.180,-55.182,-178.853,6.605,148.874
C05149=1157.696,124.931,-55.162,-178.856,6.603,148.874
C05150=1157.700,124.682,-55.143,-178.859,6.602,148.875
C05151=1157.706,124.433,-55.124,-178.861,6.601,148.875
C05152=1157.710,124.184,-55.103,-178.864,6.599,148.876
C05153=1157.715,123.934,-55.084,-178.866,6.598,148.876
C05154=1157.720,123.685,-55.064,-178.869,6.596,148.877
C05155=1157.725,123.436,-55.045,-178.872,6.594,148.877
C05156=1157.730,123.186,-55.025,-178.874,6.592,148.877
C05157=1157.734,122.938,-55.006,-178.877,6.591,148.878
C05158=1157.739,122.689,-54.986,-178.880,6.589,148.878
C05159=1157.743,122.439,-54.966,-178.883,6.588,148.879
C05160=1157.749,122.190,-54.947,-178.886,6.586,148.879
C05161=1157.753,121.941,-54.927,-178.889,6.584,148.880
C05162=1157.758,121.691,-54.908,-178.891,6.583,148.880
C05163=1157.763,121.443,-54.889,-178.893,6.582,148.880
C05164=1157.767,121.193,-54.869,-178.896,6.580,148.881
C05165=1157.773,120.944,-54.850,-178.899,6.578,148.881
C05166=1157.778,120.695,-54.831,-178.902,6.577,148.882
C05167=1157.782,120.445,-54.811,-178.905,6.575,148.882
C05168=1157.787,120.196,-54.792,-178.907,6.573,148.883
C05169=1157.792,119.947,-54.772,-178.910,6.572,148.883
C05170=1157.797,119.698,-54.753,-178.913,6.570,148.883
C05171=1157.801,119.449,-54.734,-178.916,6.568,148.884
C05172=1157.806,119.200,-54.715,-178.918,6.568,148.884
C05173=1157.811,118.950,-54.695,-178.921,6.566,148.885
C05174=1157.816,118.701,-54.676,-178.924,6.564,148.885
C05175=1157.820,118.452,-54.657,-178.926,6.563,148.886
C05176=1157.825,118.203,-54.637,-178.929,6.561,148.886
C05177=1157.831,117.954,-54.618,-178.932,6.559,148.886
C05178=1157.835,117.705,-54.599,-178.934,6.557,148.887
C05179=1157.840,117.456,-54.580,-178.938,6.556,148.887
C05180=1157.845,117.205,-54.561,-178.940,6.555,148.888
C05181=1157.850,116.957,-54.542,-178.943,6.554,148.888
C05182=1157.854,116.707,-54.522,-178.945,6.552,148.889
C05183=1157.860,116.459,-54.503,-178.948,6.550,148.889
C05184=1157.864,116.209,-54.484,-178.951,6.548,148.890
C05185=1157.869,115.960,-54.465,-178.954,6.547,148.890
C05186=1157.874,115.710,-54.446,-178.957,6.545,148.891
C05187=1157.879,115.462,-54.427,-178.959,6.544,148.891
C05188=1157.883,115.212,-54.407,-178.961,6.543,148.891
C05189=1157.889,114.963,-54.388,-178.964,6.541,148.892
C05190=1157.893,114.714,-54.369,-178.967,6.539,148.892
C05191=1157.898,114.464,-54.350,-178.970,6.538,148.893
C05192=1157.902,114.215,-54.331,-178.973,6.536,148.893
C05193=1157.908,113.966,-54.312,-178.976,6.535,148.894
C05194=1157.912,113.717,-54.293,-178.978,6.533,148.894
C05195=1157.917,113.468,-54.274,-178.980,6.532,148.894
C05196=1157.922,113.218,-54.255,-178.984,6.531,148.895
C05197=1157.927,112.969,-54.236,-178.986,6.529,148.895
C05198=1157.932,112.719,-54.217,-178.989,6.527,148.896
C05199=1157.936,112.471,-54.198,-178.992,6.525,148.896
C05200=1157.941,112.221,-54.179,-178.994,6.524,148.897
C05201=1157.946,111.972,-54.161,-178.997,6.523,148.897
C05202=1157.951,111.723,-54.141,-179.000,6.522,148.898
C05203=1157.955,111.474,-54.122,-179.003,6.520,148.898
C05204=1157.961,111.224,-54.104,-179.005,6.518,148.899
C05205=1157.965,110.975,-54.085,-179.008,6.516,148.899
C05206=1157.971,110.726,-54.066,-179.011,6.515,148.899
C05207=1157.975,110.477,-54.048,-179.013,6.514,148.900
C05208=1157.980,110.227,-54.028,-179.016,6.512,148.900
C05209=1157.985,109.978,-54.010,-179.019,6.511,148.901
C05210=1157.990,109.729,-53.990,-179.021,6.509,148.901
C05211=1157.995,109.480,-53.972,-179.025,6.508,148.902
C05212=1158.000,109.231,-53.953,-179.027,6.507,148.902
C05213=1158.004,108.981,-53.935,-179.030,6.505,148.903
C05214=1158.009,108.732,-53.916,-179.032,6.503,148.903
C05215=1158.014,108.482,-53.897,-179.035,6.502,148.903
C05216=1158.019,108.234,-53.878,-179.038,6.500,148.904
C05217=1158.024,107.984,-53.860,-179.040,6.499,148.905
C05218=1158.028,107.735,-53.841,-179.043,6.498,148.905
C05219=1158.033,107.486,-53.823,-179.046,6.496,148.905
C05220=1158.038,107.237,-53.803,-179.048,6.494,148.906
C05221=1158.043,106.987,-53.785,-179.052,6.493,148.906
C05222=1158.047,106.738,-53.766,-179.054,6.492,148.907
C05223=1158.053,106.489,-53.748,-179.057,6.490,148.907
C05224=1158.057,106.220,-53.728,-179.060,6.489,148.908
C05225=1158.063,105.952,-53.707,-179.062,6.487,148.908
C05226=1158.068,105.684,-53.688,-179.065,6.486,148.909
C05227=1158.074,105.415,-53.668,-179.068,6.484,148.909
C05228=1158.078,105.166,-53.649,-179.071,6.483,148.910
C05229=1158.083,104.917,-53.631,-179.074,6.481,148.910
C05230=1158.088,104.667,-53.612,-179.077,6.479,148.911
C05231=1158.092,104.418,-53.593,-179.079,6.479,148.911
C05232=1158.097,104.169,-53.575,-179.082,6.477,148.912
C05233=1158.103,103.919,-53.557,-179.085,6.475,148.912
C05234=1158.108,103.671,-53.538,-179.087,6.474,148.912
C05235=1158.112,103.421,-53.520,-179.091,6.472,148.913
C05236=1158.117,103.172,-53.502,-179.093,6.471,148.913
C05237=1158.122,102.923,-53.482,-179.095,6.470,148.914
C05238=1158.127,102.674,-53.464,-179.098,6.468,148.914
C05239=1158.131,102.424,-53.446,-179.101,6.467,148.915
C05240=1158.136,102.175,-53.428,-179.103,6.466,148.915
C05241=1158.142,101.925,-53.409,-179.106,6.464,148.916
C05242=1158.147,101.677,-53.391,-179.109,6.462,148.916
C05243=1158.151,101.427,-53.372,-179.112,6.461,148.917
C05244=1158.156,101.177,-53.354,-179.114,6.460,148.917
C05245=1158.161,100.928,-53.336,-179.117,6.458,148.918
C05246=1158.166,100.679,-53.318,-179.120,6.457,148.918
C05247=1158.170,100.430,-53.299,-179.123,6.455,148.919
C05248=1158.175,100.180,-53.281,-179.125,6.454,148.919
C05249=1158.180,99.931,-53.263,-179.128,6.453,148.920
C05250=1158.185,99.682,-53.245,-179.130,6.451,148.920
C05251=1158.191,99.433,-53.226,-179.134,6.450,148.921
C05252=1158.195,99.183,-53.208,-179.136,6.449,148.921
C05253=1158.200,98.933,-53.190,-179.139,6.447,148.921
C05254=1158.205,98.685,-53.171,-179.141,6.445,148.922
C05255=1158.210,98.436,-53.153,-179.144,6.444,148.922
C05256=1158.214,98.187,-53.135,-179.147,6.443,148.923
C05257=1158.219,97.937,-53.117,-179.149,6.442,148.923
C05258=1158.224,97.688,-53.099,-179.152,6.440,148.924
C05259=1158.229,97.438,-53.080,-179.155,6.439,148.924
C05260=1158.234,97.189,-53.062,-179.157,6.438,148.925
C05261=1158.239,96.940,-53.044,-179.160,6.436,148.925
C05262=1158.244,96.691,-53.026,-179.163,6.435,148.926
C05263=1158.249,96.441,-53.008,-179.166,6.434,148.926
C05264=1158.253,96.191,-52.990,-179.168,6.432,148.927
C05265=1158.258,95.942,-52.972,-179.171,6.430,148.927
C05266=1158.263,95.693,-52.954,-179.174,6.429,148.928
C05267=1158.268,95.444,-52.936,-179.176,6.428,148.928
C05268=1158.273,95.195,-52.918,-179.179,6.426,148.929
C05269=1158.278,94.946,-52.900,-179.182,6.425,148.929
C05270=1158.283,94.696,-52.882,-179.184,6.424,148.930
C05271=1158.288,94.447,-52.864,-179.187,6.423,148.930
C05272=1158.292,94.197,-52.846,-179.190,6.421,148.930
C05273=1158.297,93.948,-52.829,-179.193,6.419,148.931
C05274=1158.302,93.698,-52.811,-179.195,6.419,148.932
C05275=1158.307,93.449,-52.793,-179.198,6.417,148.932
C05276=1158.312,93.200,-52.775,-179.201,6.415,148.932
C05277=1158.317,92.951,-52.757,-179.203,6.415,148.933
C05278=1158.322,92.702,-52.739,-179.206,6.413,148.933
C05279=1158.327,92.453,-52.721,-179.209,6.411,148.934
C05280=1158.332,92.203,-52.704,-179.211,6.411,148.934
C05281=1158.337,91.954,-52.686,-179.214,6.409,148.935
C05282=1158.342,91.704,-52.668,-179.217,6.407,148.935
C05283=1158.347,91.455,-52.650,-179.220,6.406,148.936
C05284=1158.351,91.205,-52.631,-179.222,6.405,148.936
C05285=1158.356,90.955,-52.614,-179.225,6.404,148.937
C05286=1158.361,90.706,-52.596,-179.228,6.402,148.937
C05287=1158.365,90.457,-52.579,-179.230,6.401,148.938
C05288=1158.370,90.208,-52.561,-179.233,6.400,148.938
C05289=1158.375,89.958,-52.543,-179.236,6.398,148.939
C05290=1158.380,89.709,-52.525,-179.238,6.397,148.939
C05291=1158.385,89.460,-52.507,-179.241,6.396,148.940
C05292=1158.390,89.211,-52.489,-179.244,6.394,148.940
C05293=1158.395,88.961,-52.472,-179.246,6.394,148.941
C05294=1158.400,88.712,-52.454,-179.249,6.392,148.941
C05295=1158.404,88.463,-52.437,-179.252,6.390,148.942
C05296=1158.410,88.213,-52.420,-179.254,6.390,148.942
C05297=1158.415,87.964,-52.402,-179.257,6.388,148.943
C05298=1158.419,87.715,-52.384,-179.260,6.386,148.943
C05299=1158.425,87.465,-52.366,-179.263,6.386,148.944
C05300=1158.430,87.216,-52.348,-179.265,6.384,148.944
C05301=1158.434,86.967,-52.331,-179.268,6.382,148.945
C05302=1158.439,86.717,-52.314,-179.270,6.381,148.945
C05303=1158.444,86.468,-52.296,-179.273,6.380,148.946
C05304=1158.449,86.218,-52.278,-179.276,6.378,148.946
C05305=1158.455,85.970,-52.261,-179.278,6.378,148.947
C05306=1158.459,85.720,-52.244,-179.281,6.376,148.947
C05307=1158.464,85.471,-52.226,-179.284,6.375,148.948
C05308=1158.469,85.222,-52.208,-179.286,6.374,148.948
C05309=1158.474,84.972,-52.191,-179.290,6.372,148.949
C05310=1158.478,84.723,-52.174,-179.292,6.371,148.949
C05311=1158.484,84.474,-52.156,-179.294,6.370,148.950
C05312=1158.488,84.224,-52.138,-179.298,6.368,148.950
C05313=1158.493,83.975,-52.122,-179.300,6.368,148.951
C05314=1158.498,83.726,-52.104,-179.303,6.366,148.951
C05315=1158.503,83.476,-52.086,-179.306,6.365,148.952
C05316=1158.508,83.227,-52.068,-179.308,6.364,148.952
C05317=1158.512,82.977,-52.052,-179.311,6.362,148.953
C05318=1158.518,82.728,-52.034,-179.314,6.361,148.953
C05319=1158.523,82.479,-52.017,-179.316,6.360,148.954
C05320=1158.528,82.230,-52.000,-179.319,6.358,148.954
C05321=1158.533,81.980,-51.982,-179.321,6.358,148.955
C05322=1158.538,81.731,-51.965,-179.324,6.356,148.955
C05323=1158.542,81.482,-51.948,-179.327,6.354,148.956
C05324=1158.547,81.232,-51.930,-179.329,6.354,148.956
C05325=1158.552,80.982,-51.913,-179.332,6.352,148.957
C05326=1158.557,80.734,-51.896,-179.335,6.352,148.957
C05327=1158.562,80.484,-51.879,-179.338,6.350,148.958
C05328=1158.568,80.215,-51.860,-179.340,6.348,148.958
C05329=1158.572,79.947,-51.842,-179.343,6.347,148.959
C05330=1158.578,79.679,-51.823,-179.346,6.346,148.959
C05331=1158.583,79.410,-51.804,-179.349,6.345,148.960
C05332=1158.588,79.161,-51.788,-179.352,6.343,148.960
C05333=1158.593,78.911,-51.770,-179.354,6.342,148.961
C05334=1158.598,78.663,-51.753,-179.357,6.341,148.961
C05335=1158.603,78.413,-51.736,-179.360,6.339,148.962
C05336=1158.608,78.164,-51.719,-179.362,6.339,148.962
C05337=1158.613,77.914,-51.702,-179.365,6.337,148.963
C05338=1158.618,77.665,-51.684,-179.367,6.336,148.963
C05339=1158.623,77.416,-51.668,-179.370,6.335,148.964
C05340=1158.628,77.166,-51.651,-179.373,6.333,148.964
C05341=1158.633,76.917,-51.634,-179.376,6.333,148.965
C05342=1158.637,76.667,-51.616,-179.379,6.331,148.965
C05343=1158.642,76.418,-51.599,-179.381,6.330,148.966
C05344=1158.648,76.169,-51.582,-179.384,6.329,148.967
C05345=1158.652,75.919,-51.566,-179.387,6.327,148.967
C05346=1158.657,75.670,-51.548,-179.389,6.326,148.967
C05347=1158.662,75.420,-51.532,-179.392,6.325,148.968
C05348=1158.667,75.172,-51.514,-179.394,6.324,148.969
C05349=1158.672,74.922,-51.497,-179.397,6.323,148.969
C05350=1158.677,74.672,-51.480,-179.399,6.322,148.970
C05351=1158.682,74.423,-51.463,-179.402,6.320,148.970
C05352=1158.687,74.174,-51.447,-179.405,6.319,148.971
C05353=1158.692,73.924,-51.430,-179.408,6.318,148.971
C05354=1158.696,73.675,-51.413,-179.410,6.316,148.972
C05355=1158.702,73.425,-51.396,-179.413,6.316,148.972
C05356=1158.707,73.176,-51.380,-179.416,6.314,148.973
C05357=1158.712,72.926,-51.362,-179.418,6.314,148.973
C05358=1158.716,72.677,-51.346,-179.421,6.312,148.974
C05359=1158.721,72.428,-51.328,-179.424,6.310,148.974
C05360=1158.726,72.179,-51.311,-179.426,6.310,148.975
C05361=1158.731,71.929,-51.295,-179.429,6.308,148.975
C05362=1158.736,71.680,-51.278,-179.431,6.307,148.976
C05363=1158.741,71.431,-51.261,-179.435,6.306,148.976
C05364=1158.746,71.181,-51.245,-179.437,6.305,148.977
C05365=1158.751,70.932,-51.227,-179.440,6.304,148.977
C05366=1158.756,70.682,-51.212,-179.442,6.303,148.978
C05367=1158.761,70.433,-51.195,-179.445,6.301,148.978
C05368=1158.766,70.183,-51.178,-179.447,6.301,148.979
C05369=1158.771,69.934,-51.161,-179.450,6.299,148.979
C05370=1158.776,69.685,-51.145,-179.453,6.298,148.980
C05371=1158.781,69.435,-51.128,-179.456,6.297,148.980
C05372=1158.786,69.186,-51.111,-179.458,6.295,148.981
C05373=1158.790,68.937,-51.095,-179.461,6.295,148.982
C05374=1158.796,68.687,-51.077,-179.464,6.293,148.982
C05375=1158.801,68.438,-51.061,-179.466,6.292,148.983
C05376=1158.805,68.189,-51.044,-179.469,6.291,148.983
C05377=1158.810,67.938,-51.028,-179.471,6.290,148.984
C05378=1158.816,67.689,-51.011,-179.474,6.288,148.984
C05379=1158.820,67.440,-50.995,-179.477,6.288,148.985
C05380=1158.825,67.191,-50.979,-179.480,6.286,148.985
C05381=1158.830,66.942,-50.962,-179.482,6.285,148.986
C05382=1158.835,66.692,-50.945,-179.485,6.284,148.986
C05383=1158.840,66.442,-50.929,-179.487,6.283,148.987
C05384=1158.845,66.193,-50.912,-179.490,6.282,148.987
C05385=1158.850,65.944,-50.896,-179.493,6.281,148.988
C05386=1158.855,65.694,-50.879,-179.495,6.279,148.988
C05387=1158.860,65.445,-50.862,-179.498,6.279,148.989
C05388=1158.865,65.195,-50.846,-179.501,6.277,148.989
C05389=1158.869,64.946,-50.830,-179.503,6.276,148.990
C05390=1158.875,64.697,-50.814,-179.506,6.275,148.991
C05391=1158.880,64.447,-50.797,-179.508,6.274,148.991
C05392=1158.885,64.197,-50.780,-179.511,6.273,148.991
C05393=1158.890,63.948,-50.764,-179.514,6.272,148.992
C05394=1158.894,63.699,-50.747,-179.516,6.270,148.992
C05395=1158.899,63.450,-50.732,-179.519,6.270,148.993
C05396=1158.904,63.200,-50.715,-179.522,6.268,148.994
C05397=1158.910,62.951,-50.698,-179.524,6.267,148.994
C05398=1158.915,62.701,-50.682,-179.527,6.266,148.995
C05399=1158.920,62.452,-50.666,-179.529,6.265,148.995
C05400=1158.924,62.203,-50.649,-179.533,6.264,148.996
C05401=1158.930,61.953,-50.634,-179.535,6.263,148.996
C05402=1158.934,61.704,-50.617,-179.538,6.262,148.997
C05403=1158.939,61.454,-50.601,-179.540,6.261,148.997
C05404=1158.944,61.205,-50.585,-179.543,6.259,148.998
C05405=1158.949,60.956,-50.568,-179.545,6.259,148.998
C05406=1158.954,60.706,-50.552,-179.548,6.257,148.999
C05407=1158.960,60.457,-50.536,-179.551,6.257,149.000
C05408=1158.964,60.207,-50.520,-179.554,6.255,149.000
C05409=1158.969,59.958,-50.503,-179.556,6.254,149.001
C05410=1158.974,59.708,-50.487,-179.559,6.253,149.001
C05411=1158.979,59.459,-50.471,-179.561,6.252,149.001
C05412=1158.984,59.209,-50.455,-179.564,6.251,149.002
C05413=1158.989,58.960,-50.439,-179.566,6.250,149.003
C05414=1158.994,58.710,-50.423,-179.569,6.249,149.003
C05415=1158.999,58.461,-50.407,-179.572,6.247,149.004
C05416=1159.004,58.211,-50.391,-179.574,6.247,149.004
C05417=1159.009,57.962,-50.374,-179.577,6.245,149.005
C05418=1159.014,57.712,-50.358,-179.579,6.244,149.005
C05419=1159.019,57.464,-50.342,-179.583,6.243,149.006
C05420=1159.024,57.214,-50.326,-179.585,6.242,149.006
C05421=1159.029,56.965,-50.310,-179.588,6.241,149.007
C05422=1159.034,56.715,-50.294,-179.590,6.240,149.007
C05423=1159.038,56.466,-50.278,-179.593,6.239,149.008
C05424=1159.044,56.216,-50.262,-179.596,6.238,149.009
C05425=1159.049,55.966,-50.246,-179.598,6.237,149.009
C05426=1159.054,55.718,-50.230,-179.601,6.236,149.010
C05427=1159.059,55.468,-50.214,-179.603,6.235,149.010
C05428=1159.064,55.218,-50.198,-179.606,6.234,149.011
C05429=1159.069,54.969,-50.182,-179.608,6.233,149.011
C05430=1159.074,54.719,-50.166,-179.612,6.232,149.012
C05431=1159.079,54.470,-50.150,-179.614,6.231,149.012
C05432=1159.084,54.202,-50.133,-179.617,6.229,149.013
C05433=1159.090,53.933,-50.116,-179.619,6.229,149.013
C05434=1159.094,53.665,-50.099,-179.622,6.227,149.014
C05435=1159.100,53.396,-50.082,-179.626,6.226,149.015
C05436=1159.105,53.147,-50.066,-179.628,6.225,149.015
C05437=1159.110,52.897,-50.050,-179.630,6.225,149.016
C05438=1159.115,52.648,-50.034,-179.633,6.223,149.016
C05439=1159.120,52.398,-50.018,-179.635,6.222,149.017
C05440=1159.125,52.148,-50.002,-179.639,6.221,149.017
C05441=1159.131,51.899,-49.987,-179.641,6.220,149.018
C05442=1159.135,51.650,-49.971,-179.644,6.219,149.018
C05443=1159.140,51.400,-49.955,-179.646,6.218,149.019
C05444=1159.145,51.151,-49.940,-179.649,6.217,149.020
C05445=1159.150,50.901,-49.924,-179.652,6.216,149.020
C05446=1159.155,50.651,-49.908,-179.654,6.215,149.021
C05447=1159.160,50.403,-49.892,-179.657,6.213,149.021
C05448=1159.165,50.153,-49.877,-179.660,6.213,149.022
C05449=1159.170,49.903,-49.861,-179.662,6.212,149.022
C05450=1159.175,49.654,-49.845,-179.664,6.210,149.023
C05451=1159.181,49.405,-49.830,-179.667,6.210,149.023
C05452=1159.185,49.154,-49.814,-179.670,6.208,149.024
C05453=1159.190,48.905,-49.799,-179.672,6.208,149.024
C05454=1159.195,48.657,-49.782,-179.675,6.207,149.025
C05455=1159.200,48.407,-49.767,-179.678,6.206,149.026
C05456=1159.205,48.157,-49.751,-179.680,6.205,149.026
C05457=1159.210,47.908,-49.736,-179.683,6.204,149.027
C05458=1159.215,47.659,-49.720,-179.685,6.203,149.027
C05459=1159.220,47.408,-49.704,-179.688,6.202,149.028
C05460=1159.225,47.159,-49.689,-179.691,6.201,149.028
C05461=1159.230,46.910,-49.674,-179.693,6.200,149.029
C05462=1159.235,46.661,-49.658,-179.696,6.199,149.029
C05463=1159.240,46.410,-49.642,-179.698,6.198,149.030
C05464=1159.245,46.161,-49.627,-179.701,6.197,149.030
C05465=1159.250,45.912,-49.612,-179.704,6.195,149.031
C05466=1159.256,45.663,-49.596,-179.706,6.195,149.032
C05467=1159.260,45.413,-49.581,-179.709,6.194,149.032
C05468=1159.265,45.163,-49.565,-179.712,6.193,149.033
C05469=1159.271,44.914,-49.549,-179.714,6.192,149.033
C05470=1159.275,44.665,-49.534,-179.717,6.191,149.034
C05471=1159.280,44.415,-49.518,-179.719,6.190,149.034
C05472=1159.285,44.165,-49.503,-179.722,6.189,149.035
C05473=1159.290,43.916,-49.488,-179.725,6.188,149.035
C05474=1159.295,43.667,-49.472,-179.727,6.187,149.036
C05475=1159.301,43.418,-49.457,-179.730,6.186,149.037
C05476=1159.305,43.168,-49.441,-179.733,6.185,149.037
C05477=1159.310,42.918,-49.426,-179.735,6.184,149.038
C05478=1159.315,42.669,-49.411,-179.738,6.184,149.038
C05479=1159.320,42.420,-49.395,-179.740,6.182,149.039
C05480=1159.326,42.170,-49.380,-179.743,6.182,149.039
C05481=1159.331,41.921,-49.365,-179.745,6.181,149.040
C05482=1159.335,41.671,-49.349,-179.748,6.179,149.040
C05483=1159.340,41.422,-49.334,-179.750,6.179,149.041
